# B&R Automation Studio project Embraco_LinkaNaOdlievanieRotorov_DokoncovaciaStanica_Rev2
Automation Studio 4.10.3.60 SP; technology packages: Acp10Arnc0 5.15.1, mapp 5.15.0

## Configuration Config1

CPU X20cPS9400, AutomationRuntime B4.91, Build 6.3.0, Safety 1.10, Vc V4.72.6

### Task classes (Cpu.sw)
```
Cyclic#1 (cycle 3000 us, tolerance 0 us):
  RychleDeje <- Program.RychleDeje.prg
  VstupnyMan <- Program.VstupnyManipulator.prg
Cyclic#2 (cycle 10000 us, tolerance 10000 us):
  RiadenieSe <- RiadenieServ.RiadenieServ.prg
  Serva_Prir <- RiadenieServ.Serva_PriradenieVstupov.prg
  StanicaVa1 <- Program.StanicaVonkajsiehoValcovania.prg
  StanicaStr <- Program.StanicaStrihania.prg
  StanicaVal <- Program.StanicaVnutornehoValcovania.prg
  StanicaMer <- Program.StanicaMerania.prg
  RiadenieMe <- RiadenieMenicov.RiadenieMenicov.prg
  Blikanie10 <- Blikace.Blikanie10ms.prg
Cyclic#3:
  Blikanie1 <- Blikace.Blikanie50ms.prg
  OtocnyStol <- Program.OtocnyStol.prg
Cyclic#4 (cycle 200000 us, tolerance 200000 us):
  Blikanie20 <- Blikace.Blikanie200ms.prg
  ZdvihRotor <- Program.ZdvihRotora.prg
Cyclic#5 (cycle 500000 us, tolerance 500000 us):
  Blikanie50 <- Blikace.Blikanie500ms.prg
Cyclic#6 (cycle 1000000 us, tolerance 1000000 us):
  Blikanie1s <- Blikace.Blikanie1s.prg
Cyclic#7 (cycle 5000000 us, tolerance 5000000 us):
  Blikanie5s <- Blikace.Blikanie5s.prg
Cyclic#8 (cycle 100000 us, tolerance 100000 us):
  VystupnyOd <- Program.VystupnyOdsuvac.prg
  StanicaRaz <- Program.StanicaRazenia.prg
  VystupnyMa <- Program.VystupnyManipulator.prg
  Oddelovac <- Program.Oddelovac.prg
  Main <- Program.Main.prg
  Komunikaci <- Komunikacia.KOM_HlavnaLinka.prg
  Poruchy_Si <- Program.Poruchy_Signalizacie.prg
DataObjects: Acp10sys, assl1
NcDataObjects: acp10etxen <- RiadenieServ.acp10etxen.dob, gAxis01a <- RiadenieServ.VstupnyManipulator.gAxis01a.dob, gAxis01i <- RiadenieServ.VstupnyManipulator.gAxis01i.dob, gAxis02a <- RiadenieServ.VystupnyManipulator.gAxis02a.dob, gAxis02i <- RiadenieServ.VystupnyManipulator.gAxis02i.dob, gAxis03a <- RiadenieServ.ZdvihValcovacky.gAxis03a.dob, gAxis03i <- RiadenieServ.ZdvihValcovacky.gAxis03i.dob, gAxis04a <- RiadenieServ.ZdvihRotora.gAxis04a.dob, gAxis04i <- RiadenieServ.ZdvihRotora.gAxis04i.dob
VcDataObjects: Visu <- Vizualizacia.Visu.dob
Binaries: udbdef, TCData, arsvcreg, vccbtn, arialbd, vcmgr, vcgclass, vcfile, vccnum, vctcal, vcdsloc, vcbclass, vcfntttf, vccalarm, arial, vcpdi815, vccshape, vcalarm, vcptelo, Visu01, vccdt, vcpdsw, vcpdihd, vcpk, vccbmp, vccstr, vcpfppc7, vcrt, vcshared, Visu02, vcctext, vcclbox, vccbar, vcpdi855, vcdsint, vccovl, vccline, Visu03, iomap, asfw, Role, ashwac, sysconf, Config_1, ashwd, Config, User, arconfig, acp10cfg, Acp10map, vcchspot
Libraries: Acp10par, NcGlobal, Acp10man, AsSafety, FileIO, DataObj, AsXml, standard, runtime, astime, AsEPL, AsIOAcc, Acp10_MC, brsystem, sys_lib, IecCheck, SC, AsBrStr, MpRecipe, MpBase, AxisLib, asieccon, powerlnk, vcresman
```

### Hardware
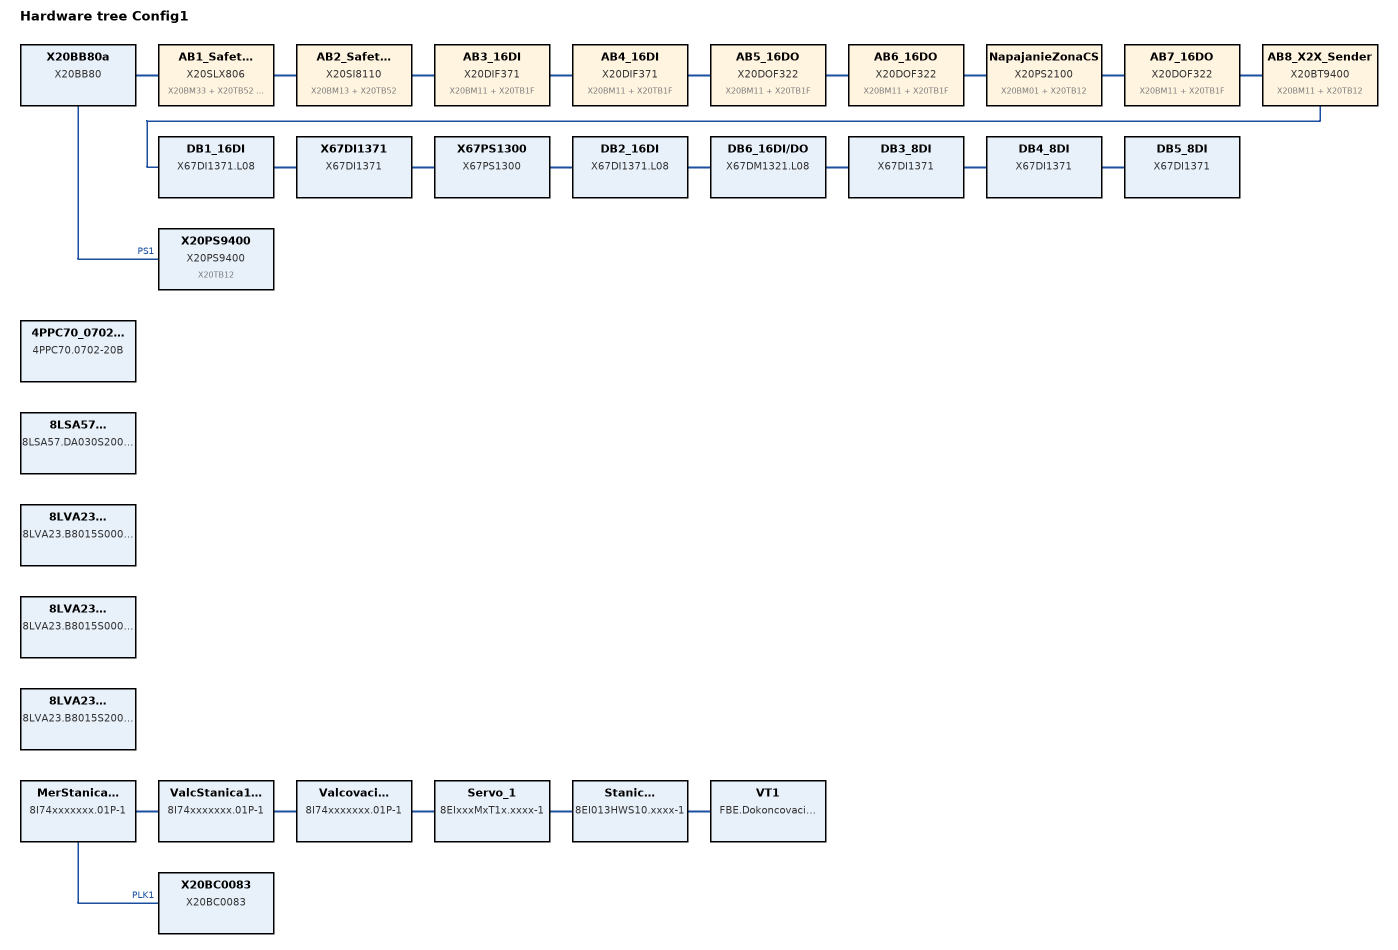
```
4PPC70_0702_20B : 4PPC70.0702-20B v1.5.4.0
  Connector IF1:
    DNAConfiguration = manual
    CycleTime = 1000
    EplNatSubnet = 192.168.100.0
  Connector IF2:
    ActivateDevice = 1
    Mode = Manual
    InternetAddress = 192.168.0.3
    SubnetMask = 255.255.255.0
    ActivateModbus = 1
    NumSlaves = -1
    NumAllBlocks = -1
    MemSizeIn = -1
    MemSizeOut = -1
    ModbusSlaveGrey = 1
    ModbusSlaveConfig_1
    InputRegisterChannelGroup1_1
    InputRegisterChannelID1_1 = OUT_1
    InputRegisterChannelType1_1 = UINT
    InputRegisterChannelGroup2_1
    InputRegisterChannelID2_1 = OUT_2
    InputRegisterChannelAddress2_1 = 8193
    InputRegisterChannelType2_1 = UINT
    InputRegisterChannelGroup3_1
    InputRegisterChannelID3_1 = OUT_3
    InputRegisterChannelAddress3_1 = 8194
    InputRegisterChannelType3_1 = UINT
    InputRegisterChannelGroup4_1
    InputRegisterChannelID4_1 = OUT_4
    InputRegisterChannelAddress4_1 = 8195
    InputRegisterChannelType4_1 = UINT
    InputRegisterChannelGroup5_1
    InputRegisterChannelID5_1 = OUT_5
    InputRegisterChannelAddress5_1 = 8196
    InputRegisterChannelType5_1 = UINT
    HoldingRegisterChannelGroup1_1
    HoldingRegisterChannelID1_1 = IN_1
    HoldingRegisterChannelType1_1 = UINT
    HoldingRegisterChannelGroup2_1
    HoldingRegisterChannelID2_1 = IN_2
    HoldingRegisterChannelAddress2_1 = 24577
    HoldingRegisterChannelType2_1 = UINT
    HoldingRegisterChannelGroup3_1
    HoldingRegisterChannelID3_1 = IN_3
    HoldingRegisterChannelAddress3_1 = 24578
    HoldingRegisterChannelType3_1 = UINT
    HoldingRegisterChannelGroup4_1
    HoldingRegisterChannelID4_1 = IN_4
    HoldingRegisterChannelAddress4_1 = 24579
    HoldingRegisterChannelType4_1 = UINT
    HoldingRegisterChannelGroup5_1
    HoldingRegisterChannelID5_1 = IN_5
    HoldingRegisterChannelAddress5_1 = 24580
    HoldingRegisterChannelType5_1 = UINT
    ModbusMaster = 0
  Connector IF5:
    CycleTime = 1000
  ConfigurationID = Embraco_LinkaNaOdlievanieRotorov_DokoncovaciaStanica_Config1
  UserPartitionSize = 0
  PermanentPvSize = 2000
  RemanentGlobalPvSize = 2000
  DisableProfiling = 1
  TimerDeviceType = EPLX2X
  TimerDevice = 4PPC70_0702_20B.IF1
  TaskClassIdleTime = 2000
  Cyclic1Duration = 3000
  Cyclic1Tolerance = 0
  Cyclic2Duration = 10000
  Cyclic2Tolerance = 10000
  Cyclic4Duration = 200000
  Cyclic4Tolerance = 200000
  Cyclic5Duration = 500000
  Cyclic5Tolerance = 500000
  Cyclic6Duration = 1000000
  Cyclic6Tolerance = 1000000
  Cyclic7Duration = 5000000
  Cyclic7Tolerance = 5000000
  Cyclic8Duration = 100000
  Cyclic8Tolerance = 100000
  FileDevice1
  FileDeviceName1 = HDD
  FileDevicePath1 = C:\
  TimeZone = 145
  FtpUser1
  FtpUsername1 = admin
  FtpUserPassword1 = kfejnbuok6+6ErbPl2VMIFPsI8vTqz8wcboRfqSMuVU=
  FtpUserSalt1 = 0YUTbZnu
  FTPAccessRight1 = 0
  FTPMSPartition1 = SYSTEM
  VcObjectName = Visu
  KeyMappingFile = VC\4PPC70_0702_20B.dis
8LSA57.DA030S200-3 : 8LSA57.DA030S200-3 v1.0.5.34  [EC -> StanicaValcovania2.EC1; MT -> StanicaValcovania2.MT1]
8LVA23.B8015S000-0 : 8LVA23.B8015S000-0 v1.0.1.30  [EC -> Servo_1.EC1; MT -> Servo_1.MT1]
8LVA23.B8015S000-0a : 8LVA23.B8015S000-0 v1.0.1.30  [EC -> Servo_1.EC2; MT -> Servo_1.MT2]
8LVA23.B8015S200-0 : 8LVA23.B8015S200-0 v2.2.0.3  [EC -> Servo_1.EC3; MT -> Servo_1.MT3]
AB1_SafetyMaster : X20SLX806 v1.10.12.1  [SS1 -> X20TB52.SS; SS2 -> X20TB52a.SS; SL -> X20BM33.SL1]
  Supervision = off
  SafeProject = SafeLOGIC-1
  SafeDesigner = 4.3.4.4
  DigitalOutput01 = viaSafeLOGIC
  DigitalOutput02 = viaSafeLOGIC
  DigitalOutput03 = viaSafeLOGIC
  DigitalOutput04 = viaSafeLOGIC
  DigitalOutput05 = viaSafeLOGIC
  DigitalOutput06 = viaSafeLOGIC
  UnsafeOutputBOOLs = 16
  UnsafeInputBOOLs = 16
AB2_SafetyInputs : X20SI8110 v1.10.12.0  [SS1 -> X20TB52b.SS; SL -> X20BM13.SL1]
  Supervision = off
AB3_16DI : X20DIF371 v1.2.0.0  [SS1 -> X20TB1F.SS; SL -> X20BM11.SL1]
  Supervision = off
AB4_16DI : X20DIF371 v1.2.0.0  [SS1 -> X20TB1F1.SS; SL -> X20BM11a.SL1]
  Supervision = off
AB5_16DO : X20DOF322 v1.5.0.0  [SS1 -> X20TB1F2.SS; SL -> X20BM11b.SL1]
  Supervision = off
AB6_16DO : X20DOF322 v1.5.0.0  [SS1 -> X20TB1F4.SS; SL -> X20BM11e.SL1]
  Supervision = off
AB7_16DO : X20DOF322 v1.5.0.0  [SS1 -> X20TB1F3.SS; SL -> X20BM11c.SL1]
  Supervision = off
AB8_X2X_Sender : X20BT9400 v1.3.0.0  [SS1 -> X20TB12b.SS; SL -> X20BM11d.SL1]
  Supervision = off
  PowerInfo = on
DB1_16DI : X67DI1371.L08 v1.1.0.0  [X2X1 -> AB8_X2X_Sender.X2X1 [Cable Type=X2XCable, Length=10, Version=1.0.0.3]]
  Supervision = off
DB2_16DI : X67DI1371.L08 v1.1.0.0  [X2X1 -> X67PS1300.X2X2 [Cable Type=X2XCable, Length=10, Version=1.0.0.3]]
  Supervision = off
DB3_8DI : X67DI1371 v1.1.0.0  [X2X1 -> DB6_16DI/DO.X2X2 [Cable Type=X2XCable, Length=10, Version=1.0.0.3]]
  Supervision = off
DB4_8DI : X67DI1371 v1.1.0.0  [X2X1 -> DB3_8DI.X2X2 [Cable Type=X2XCable, Length=10, Version=1.0.0.3]]
  Supervision = off
DB5_8DI : X67DI1371 v1.1.0.0  [X2X1 -> DB4_8DI.X2X2 [Cable Type=X2XCable, Length=10, Version=1.0.0.3]]
  Supervision = off
DB6_16DI/DO : X67DM1321.L08 v1.3.0.0  [X2X1 -> DB2_16DI.X2X2 [Cable Type=X2XCable, Length=10, Version=1.0.0.3]]
  Supervision = off
  Direction14 = output
  Direction15 = output
  Direction16 = output
MerStanica_OtacanieRotora : 8I74xxxxxxx.01P-1 v1.6.2.0  [PLK1 -> X20BC0083.PLK1 [Cable Type=PowerlinkCable, Length=10, Version=1.0.0.3]; PLK2 -> ValcStanica1_OtacanieRotora.PLK1 [Cable Type=PowerlinkCable, Length=10, Version=1.0.0.3]]
  FunctionModel = Standard
  Supervision = off
  LFRD_LFR_Filter = LFR_RFR
  ACC = 10
  DEC = 10
  CTT = 0
  NPR = 25
  COS = 77
  UNS = 230
  NCR = 13
  NSP = 1380
  PTCL = 1
NapajanieZonaCS : X20PS2100 v1.4.0.0  [SS1 -> X20TB12a.SS; SL -> X20BM01.SL1]
  Supervision = off
  PowerInfo = on
Servo_1 : 8EIxxxMxT1x.xxxx-1 v2.3.1.1  [PLK1 -> ValcovaciaStanica2_OtacanieNastroja.PLK2 (NodeNumber=4) [Cable Type=PowerlinkCable, Length=10, Version=1.0.0.3]; PLK2 -> StanicaValcovania2.PLK1 (NodeNumber=4) [Cable Type=PowerlinkCable, Length=10, Version=1.0.0.3]; EC1 -> 8LVA23.B8015S000-0.EC; EC2 -> 8LVA23.B8015S000-0a.EC; EC3 -> 8LVA23.B8015S200-0.EC; MT2 -> 8LVA23.B8015S000-0a.MT; MT3 -> 8LVA23.B8015S200-0.MT]
  BothEndSwitchesAreNormallyOpen_r1 = on
  QuickStopIsNormallyOpen_r1 = on
  BothEndSwitchesAreNormallyOpen_r2 = on
  QuickStopIsNormallyOpen_r2 = on
  BothEndSwitchesAreNormallyOpen_r3 = on
  QuickStopIsNormallyOpen_r3 = on
  Ax1Interface = Ax1EnDat
  Ax2Interface = Ax2EnDat
  Ax3Interface = Ax3EnDat
StanicaValcovania2 : 8EI013HWS10.xxxx-1 v2.3.1.1  [PLK1 -> Servo_1.PLK2 (NodeNumber=7) [Cable Type=PowerlinkCable, Length=10, Version=1.0.0.3]; PLK2 -> VT1.PLK1 (NodeNumber=7) [Cable Type=PowerlinkCable, Length=10, Version=1.0.0.3]; EC1 -> 8LSA57.DA030S200-3.EC]
  MotionTP = Acp10Arnc0
  BothEndSwitchesAreNormallyOpen_r1 = on
  QuickStopIsNormallyOpen_r1 = on
  Ax1Interface = Ax1EnDat
VT1 : FBE.DokoncovaciaStanica_VT1 v11.13.09 (OrderNumber=VT1)  [PLK1 -> StanicaValcovania2.PLK2 (NodeNumber=5) [Cable Type=PowerlinkCable, Length=10, Version=1.0.0.3]]
  Supervision = off
  p2000s01_direction = wo
  p2000s02_direction = wo
  p2000s03_direction = wo
  p2000s04_direction = wo
ValcStanica1_OtacanieRotora : 8I74xxxxxxx.01P-1 v1.6.2.0  [PLK1 -> MerStanica_OtacanieRotora.PLK2 [Cable Type=PowerlinkCable, Length=10, Version=1.0.0.3]; PLK2 -> ValcovaciaStanica2_OtacanieNastroja.PLK1 [Cable Type=PowerlinkCable, Length=10, Version=1.0.0.3]]
  FunctionModel = Standard
  Supervision = off
  LFRD_LFR_Filter = LFR_RFR
  ACC = 10
  DEC = 10
  CTT = 0
  NPR = 150
  COS = 79
  UNS = 230
  NCR = 56
  NSP = 1415
  PTCL = 1
ValcovaciaStanica2_OtacanieNastroja : 8I74xxxxxxx.01P-1 v1.6.2.0  [PLK1 -> ValcStanica1_OtacanieRotora.PLK2 (NodeNumber=6) [Cable Type=PowerlinkCable, Length=10, Version=1.0.0.3]; PLK2 -> Servo_1.PLK1 (NodeNumber=6) [Cable Type=PowerlinkCable, Length=10, Version=1.0.0.3]]
  FunctionModel = Standard
  Supervision = off
  LFRD_LFR_Filter = LFR_RFR
  ACC = 40
  DEC = 40
  CTT = 0
  NPR = 110
  COS = 84
  UNS = 400
  NCR = 25
  NSP = 2825
  BLC = 2
  PTCL = 1
X20BB80a : X20BB80 v1.1.0.0
X20BC0083 : X20BC0083 v2.14.0.0  [PLK1 -> MerStanica_OtacanieRotora.PLK1 [Cable Type=PowerlinkCable, Length=10, Version=1.0.0.3]; PLK2 -> 4PPC70_0702_20B.IF1 [Cable Type=PowerlinkCable, Length=10, Version=1.0.0.3]; SL -> X20BB80a.SL1]
  Supervision = off
X20BM01 : X20BM01 v2.2.0.0  [X2X1 -> X20BM11e.X2X2]
X20BM11 : X20BM11 v1.1.0.0  [X2X1 -> X20BM13.X2X2]
X20BM11a : X20BM11 v1.1.0.0  [X2X1 -> X20BM11.X2X2]
X20BM11b : X20BM11 v1.1.0.0  [X2X1 -> X20BM11a.X2X2]
X20BM11c : X20BM11 v1.1.0.0  [X2X1 -> X20BM01.X2X2]
X20BM11d : X20BM11 v1.1.0.0  [X2X1 -> X20BM11c.X2X2]
X20BM11e : X20BM11 v1.1.0.0  [X2X1 -> X20BM11b.X2X2]
X20BM13 : X20BM13 v1.1.0.0  [X2X1 -> X20BM33.X2X2]
X20BM33 : X20BM33 v1.1.0.0  [X2X1 -> X20BB80a.IF1]
X20PS9400 : X20PS9400 v1.7.0.0  [SS1 -> X20TB12c.SS; PS -> X20BB80a.PS1]
  Supervision = off
  PowerInfo = on
X20TB12a : X20TB12 v1.0.0.0
X20TB12b : X20TB12 v1.0.0.0
X20TB12c : X20TB12 v1.0.0.0
X20TB1F : X20TB1F v1.0.0.0
X20TB1F1 : X20TB1F v1.0.0.0
X20TB1F2 : X20TB1F v1.0.0.0
X20TB1F3 : X20TB1F v1.0.0.0
X20TB1F4 : X20TB1F v1.0.0.0
X20TB52 : X20TB52 v1.0.0.2
X20TB52a : X20TB52 v1.0.0.2
X20TB52b : X20TB52 v1.0.0.2
X67DI1371 : X67DI1371 v1.1.0.0  [X2X1 -> DB1_16DI.X2X2 [Cable Type=X2XCable, Length=10, Version=1.0.0.3]]
  Supervision = off
X67PS1300 : X67PS1300 v1.0.0.0  [X2X1 -> X67DI1371.X2X2 [Cable Type=X2XCable, Length=10, Version=1.0.0.3]]
```

### Cpu.per - 4PPC70_0702_20B/Cpu.per
```iecst
VAR_CONFIG
	Valcovanie_RychlostJog_MM_s AT %MD0; (* *)
	VstupManipul_RychlostJog_MM_s AT %MD4; (* *)
	VystupManipul_RychlostJog_MM_s AT %MD8; (* *)
	Stol_Pozicia_1 AT %MB12; (*Pozicia stola pod meranim  0 - neznamy kus, 1 - kus OK, 2 - kus NG *)
	Stol_Pozicia_2 AT %MB13; (*Pozícia medzi meranim a výstupným manipulátorom    0 - neznamy kus, 1 - kus OK, 2 - kus NG *)
	Stol_Pozicia_3 AT %MB14; (*Pozícia pod výstupným manipulátorom     0 - neznamy kus, 1 - kus OK, 2 - kus NG *)
	TP_Meranie_CasMerania AT %MD16; (*v s*)
	TP_Meranie_RychlostOtacania AT %MW20; (*v Hz*)
	TP_Razenie_CasRazenia AT %MD24; (*v s*)
	TP_Valcovanie_PoziciaVnorenia AT %MD28; (*v mm*)
	TP_Valcovanie_RychlostOtacania AT %MW32; (*v Hz*)
	TP_Valcovanie_RychlostZdvihu AT %MD36; (*v mm/s*)
	TP_VstupManip_PoziciaOdoberania AT %MD40; (*v mm*)
	TP_VstupManip_PoziciaUkladania AT %MD44; (*v mm*)
	TP_VstupManip_RychlostPojazdu AT %MD48; (*v mm/s*)
	TP_VystupManip_PoziciaOdoberania AT %MD52; (*v mm*)
	TP_VystupManip_PoziciaUklad_NG AT %MD56; (*v mm*)
	TP_VystupManip_PoziciaUklad_OK AT %MD60; (*v mm*)
	TP_VystupManip_RychlostPojazdu AT %MD64; (*v mm/s*)
	TP_Valcovanie_CasStrekuOleja AT %MD68; (*v s*)
	TP_Valcovanie_PocetCyklPredStrek AT %MW72; (* *)
	VstupManipulator_Drzi_NG_Kus AT %MX74; (* *)
	TP_CasValcovania_s AT %MD76; (*v sek*)
	Valcovanie2_CasValcovania_s AT %MD80; (* *)
	Valcovanie2_FM_DobehRampa_s AT %MD84; (* *)
	Valcovanie2_FM_RozbehRampa_s AT %MD88; (* *)
	Valcovanie2_FM_RychlostOtac_Hz AT %MD92; (* *)
	Valcovanie2_ServoJoggRychl_MM_s AT %MD96; (* *)
	Valcovanie2_ServoPracRychl1_MM_s AT %MD100; (* *)
	Valcovanie2_ServoPracRychl2_MM_s AT %MD104; (* *)
	Valcovanie2_CasStrekuOleja_s AT %MD108; (* *)
	Valcovanie2_MomentPritlaku_Nm AT %MD112; (* *)
	Valcovanie2_PocetCyklStrekuOleja AT %MB116; (* *)
	Valcovanie2_ZadanaPozMM AT %MD120; (* *)
	Valcovanie2_ZadanaPozSTART_MM AT %MD124; (*Čakacia pozícia pod stolom*)
END_VAR
```

### IoMap.iom - 4PPC70_0702_20B/IoMap.iom
```iecst
VAR_CONFIG
	Cyclic#1.siCS_KanalA AT %IX."AB1_SafetyMaster".SafeDigitalInput01;
	Cyclic#1.siCS_KanalB AT %IX."AB1_SafetyMaster".SafeDigitalInput02;
	Cyclic#1.siServisneDvere1_KanalA AT %IX."AB1_SafetyMaster".SafeDigitalInput03;
	Cyclic#1.siServisneDvere1_KanalB AT %IX."AB1_SafetyMaster".SafeDigitalInput04;
	Cyclic#1.siServisneDvere2_KanalA AT %IX."AB1_SafetyMaster".SafeDigitalInput05;
	Cyclic#1.siServisneDvere2_KanalB AT %IX."AB1_SafetyMaster".SafeDigitalInput06;
	Cyclic#1.siServisneDvere3_KanalA AT %IX."AB1_SafetyMaster".SafeDigitalInput07;
	Cyclic#1.siServisneDvere3_KanalB AT %IX."AB1_SafetyMaster".SafeDigitalInput08;
	Cyclic#1.siServisneDvere4_KanalA AT %IX."AB2_SafetyInputs".SafeDigitalInput01;
	Cyclic#1.siServisneDvere4_KanalB AT %IX."AB2_SafetyInputs".SafeDigitalInput02;
	Cyclic#1.siServisneDvere5_KanalA AT %IX."AB2_SafetyInputs".SafeDigitalInput03;
	Cyclic#1.siServisneDvere5_KanalB AT %IX."AB2_SafetyInputs".SafeDigitalInput04;
	Cyclic#1.soMotory AT %IX."AB1_SafetyMaster".PhysicalStateChannel01;
	Cyclic#1.soVystupy AT %IX."AB1_SafetyMaster".PhysicalStateChannel02;
	Cyclic#1.soKomunikacia_StavCS AT %IX."AB1_SafetyMaster".PhysicalStateChannel03;
	Cyclic#1.Reset_CS AT %QX."AB1_SafetyMaster".BOOL101;
	Cyclic#1.Reset_Oplotenia AT %QX."AB1_SafetyMaster".BOOL102;
	Cyclic#1.Stav_BZ5_Zamknuty AT %IX."AB1_SafetyMaster".BOOL007;
	Cyclic#1.Stav_BZ4_Zamknuty AT %IX."AB1_SafetyMaster".BOOL006;
	Cyclic#1.Stav_BZ3_Zamknuty AT %IX."AB1_SafetyMaster".BOOL005;
	Cyclic#1.Stav_BZ2_Zamknuty AT %IX."AB1_SafetyMaster".BOOL004;
	Cyclic#1.Stav_BZ1_Zamknuty AT %IX."AB1_SafetyMaster".BOOL003;
	Cyclic#1.Stav_CS_Odblokovane AT %IX."AB1_SafetyMaster".BOOL002;
	Cyclic#1.SafetyPLC_Nabehlo AT %IX."AB1_SafetyMaster".BOOL001;
	Cyclic#1.diStav_PrivodVzduchuKanalA AT %QX."AB1_SafetyMaster".BOOL103;
	Cyclic#1.diStav_PrivodVzduchuKanalB AT %QX."AB1_SafetyMaster".BOOL104;
	Cyclic#1.diStavReleKA100_KA101 AT %QX."AB1_SafetyMaster".BOOL105;
	Cyclic#1.diStavReleKA102_KA103 AT %QX."AB1_SafetyMaster".BOOL106;
	Cyclic#1.diStavReleKA104_KA105 AT %QX."AB1_SafetyMaster".BOOL107;
	Cyclic#1.BezpOkruhOplotenia_Aktivovany AT %IX."AB1_SafetyMaster".BOOL010;
	Cyclic#1.BezpOkruhCS_Aktivovany AT %IX."AB1_SafetyMaster".BOOL009;
	Cyclic#1.Stav_BZ6_Zamknuty AT %IX."AB1_SafetyMaster".BOOL008;
	Cyclic#1.siServisneDvere6_KanalA AT %IX."AB2_SafetyInputs".SafeDigitalInput05;
	Cyclic#1.siServisneDvere6_KanalB AT %IX."AB2_SafetyInputs".SafeDigitalInput06;
	Cyclic#1.diMeranie_PoruchaOtacRotora AT %IX."AB3_16DI".DigitalInput01;
	Cyclic#1.diValcovanie_PoruchaOtacRotora AT %IX."AB3_16DI".DigitalInput02;
	Cyclic#1.diStol_PoruchaOtacStola AT %IX."AB3_16DI".DigitalInput03;
	Cyclic#1.diStol_TeplotaMotoraOK AT %IX."AB3_16DI".DigitalInput04;
	Cyclic#1.diPoruchaNapajaniaSERVO1 AT %IX."AB3_16DI".DigitalInput05;
	Cyclic#1.diHydraulika_PoruchaCerpadla AT %IX."AB3_16DI".DigitalInput06;
	Cyclic#1.diBZ1_DvereZavrete AT %IX."AB3_16DI".DigitalInput09;
	Cyclic#1.diBZ2_DvereZavrete AT %IX."AB3_16DI".DigitalInput10;
	Cyclic#1.diBZ3_DvereZavrete AT %IX."AB3_16DI".DigitalInput11;
	Cyclic#1.diBZ4_DvereZavrete AT %IX."AB3_16DI".DigitalInput12;
	Cyclic#1.diBZ5_DvereZavrete AT %IX."AB3_16DI".DigitalInput13;
	Cyclic#1.diStavReleKA100_KA101 AT %IX."AB3_16DI".DigitalInput14;
	Cyclic#1.diStavReleKA102_KA103 AT %IX."AB3_16DI".DigitalInput15;
	Cyclic#1.diStavReleKA104_KA105 AT %IX."AB3_16DI".DigitalInput16;
	Cyclic#1.diStav_PrivodVzduchuKanalA AT %IX."AB4_16DI".DigitalInput01;
	Cyclic#1.diStav_PrivodVzduchuKanalB AT %IX."AB4_16DI".DigitalInput02;
	Cyclic#1.diBZ6_DvereZavrete AT %IX."AB4_16DI".DigitalInput03;
	Cyclic#1.doHydraulika_ChodCerpadla AT %QX."AB5_16DO".DigitalOutput01;
	Cyclic#1.doBZ1_ZamkniZamok AT %QX."AB5_16DO".DigitalOutput02;
	Cyclic#1.doBZ2_ZamkniZamok AT %QX."AB5_16DO".DigitalOutput03;
	Cyclic#1.doBZ3_ZamkniZamok AT %QX."AB5_16DO".DigitalOutput04;
	Cyclic#1.doBZ4_ZamkniZamok AT %QX."AB5_16DO".DigitalOutput05;
	Cyclic#1.doBZ5_ZamkniZamok AT %QX."AB5_16DO".DigitalOutput06;
	Cyclic#1.doValcovanie_DavkaOleja AT %QX."AB5_16DO".DigitalOutput07;
	Cyclic#1.doKontrolkaPORUCHA AT %QX."AB5_16DO".DigitalOutput08;
	Cyclic#1.doMajak_CerveneSvetlo AT %QX."AB5_16DO".DigitalOutput09;
	Cyclic#1.doMajak_ZlteSvetlo AT %QX."AB5_16DO".DigitalOutput10;
	Cyclic#1.doMajak_ZeleneSvetlo AT %QX."AB5_16DO".DigitalOutput11;
	Cyclic#1.doMajak_Hukacka AT %QX."AB5_16DO".DigitalOutput12;
	Cyclic#1.doStol_ResetPoruchy AT %QX."AB5_16DO".DigitalOutput13;
	Cyclic#1.doBZ6_ZamkniZamok AT %QX."AB5_16DO".DigitalOutput14;
	Cyclic#1.doRazenie_ZdvihRotora AT %QX."AB7_16DO".DigitalOutput01;
	Cyclic#1.doRazenie_ZostupRotora AT %QX."AB7_16DO".DigitalOutput02;
	Cyclic#1.Vyrazanie.OUT.VyrazanieVysunut AT %QX."AB7_16DO".DigitalOutput03;
	Cyclic#1.Vyrazanie.OUT.VyrazanieZasunut AT %QX."AB7_16DO".DigitalOutput04;
	Cyclic#1.doStol_OtacajVPRED AT %QX."AB7_16DO".DigitalOutput05;
	Cyclic#1.doStol_OtacajVZAD AT %QX."AB7_16DO".DigitalOutput06;
	Cyclic#1.doStol_ODBRZDENIE AT %QX."AB7_16DO".DigitalOutput07;
	Cyclic#1.diStol_SnimacPolohyStola AT %IX."DB1_16DI".DigitalInput01;
	Cyclic#1.Vyrazanie.IN.KusPritomny AT %IX."DB1_16DI".DigitalInput02;
	Cyclic#1.Vyrazanie.IN.VyrazanieJeDole AT %IX."DB1_16DI".DigitalInput03;
	Cyclic#1.Vyrazanie.IN.VyrazanieJeHore AT %IX."DB1_16DI".DigitalInput04;
	Cyclic#1.Vyrazanie.IN.CentrovanieZatvorene AT %IX."DB1_16DI".DigitalInput05;
	Cyclic#1.Vyrazanie.IN.CentrovanieOtvorene AT %IX."DB1_16DI".DigitalInput06;
	Cyclic#1.Vyrazanie.IN.UchytenieKolikaDrzimkus AT %IX."DB1_16DI".DigitalInput07;
	Cyclic#1.Vyrazanie.IN.UchytenieNaliatkuDrzimkus AT %IX."DB1_16DI".DigitalInput08;
	Cyclic#1.Vyrazanie.IN.OdhadzovanieJeVzadu AT %IX."DB1_16DI".DigitalInput09;
	Cyclic#1.Vyrazanie.IN.OdhadzovanieJeVpredu AT %IX."DB1_16DI".DigitalInput10;
	Cyclic#1.diRazenie_ZdvihSpodnaPoloha AT %IX."DB1_16DI".DigitalInput11;
	Cyclic#1.diValcovanie_PritomnostRotora AT %IX."DB2_16DI".DigitalInput03;
	Cyclic#1.diValcovanie_GriperOtvoreny AT %IX."DB2_16DI".DigitalInput04;
	Cyclic#1.diValcovanie_GriperZatvoreny AT %IX."DB2_16DI".DigitalInput05;
	Cyclic#1.diValcovanie_HladinaOlejaOK AT %IX."DB2_16DI".DigitalInput06;
	Cyclic#1.diMeranie_ZdvihSpodnaPoloha AT %IX."DB2_16DI".DigitalInput09;
	Cyclic#1.diMeranie_ZdvihHornaPoloha AT %IX."DB2_16DI".DigitalInput10;
	Cyclic#1.diMeranie_PritomnostRotora AT %IX."DB2_16DI".DigitalInput11;
	Cyclic#1.diStol_PritomnostRotoraVstup AT %IX."DB2_16DI".DigitalInput15;
	Cyclic#1.diStol_PritomnostRotoraVystup AT %IX."DB2_16DI".DigitalInput16;
	Cyclic#1.diVstupManipul_ZasunutyHore AT %IX."DB3_8DI".DigitalInput01;
	Cyclic#1.diVstupManipul_VysunutyDole AT %IX."DB3_8DI".DigitalInput02;
	Cyclic#1.diVstupManipul_PrednyLimitSnimac AT %IX."DB3_8DI".DigitalInput03 INVERSE;
	Cyclic#1.diVstupManipul_ZadnyLimitSnimac AT %IX."DB3_8DI".DigitalInput04 INVERSE;
	Cyclic#1.diVystupManipul_ZasunutyHore AT %IX."DB4_8DI".DigitalInput01;
	Cyclic#1.diVystupManipul_PrednyLimSnimac AT %IX."DB4_8DI".DigitalInput03 INVERSE;
	Cyclic#1.diVystupManipul_ZadnyLimSnimac AT %IX."DB4_8DI".DigitalInput04 INVERSE;
	Cyclic#1.doOddelovac_PrepniPozNavazania AT %QX."VT1".Valve_1_C14;
	Cyclic#1.doOddelovac_PrepniPozVyvazania AT %QX."VT1".Valve_1_C12;
	Cyclic#1.doVystupManipul_GriperZATVOR AT %QX."VT1".Valve_5_C14;
	Cyclic#1.doVystupManipul_GriperOTVOR AT %QX."VT1".Valve_5_C12;
	Cyclic#1.doVystDopr_OdsuvacVYSUN AT %QX."VT1".Valve_6_C14;
	Cyclic#1.doVystDopr_OdsuvacZASUN AT %QX."VT1".Valve_6_C12;
	Cyclic#1.Vyrazanie.OUT.OdhadzovanieVysunut AT %QX."VT1".Valve_9_C14;
	Cyclic#1.Vyrazanie.OUT.OdhadzovanieZasunut AT %QX."VT1".Valve_9_C12;
	Cyclic#1.::FM_Menic[1].IO.ModuleOk AT %IX."MerStanica_OtacanieRotora".ModuleOk;
	Cyclic#1.::FM_Menic[1].IO.ReadyToSwitchOn AT %IX."MerStanica_OtacanieRotora".ETAD_Input_Bool_00;
	Cyclic#1.::FM_Menic[1].IO.SwitchedOn AT %IX."MerStanica_OtacanieRotora".ETAD_Input_Bool_01;
	Cyclic#1.::FM_Menic[1].IO.Running AT %IX."MerStanica_OtacanieRotora".ETAD_Input_Bool_02;
	Cyclic#1.::FM_Menic[1].IO.Fault AT %IX."MerStanica_OtacanieRotora".ETAD_Input_Bool_03;
	Cyclic#1.::FM_Menic[1].IO.VoltageEnabled AT %IX."MerStanica_OtacanieRotora".ETAD_Input_Bool_04;
	Cyclic#1.::FM_Menic[1].IO.SwitchOnDisabled AT %IX."MerStanica_OtacanieRotora".ETAD_Input_Bool_06;
	Cyclic#1.::FM_Menic[1].IO.StavRiadeniaMenica AT %IX."MerStanica_OtacanieRotora".ETAD_Input_Bool_09;
	Cyclic#1.::FM_Menic[1].IO.PoziciaDosiahnuta AT %IX."MerStanica_OtacanieRotora".ETAD_Input_Bool_10;
	Cyclic#1.::FM_Menic[1].IO.SmerOtacania AT %IX."MerStanica_OtacanieRotora".ETAD_Input_Bool_15;
	Cyclic#1.::FM_Menic[1].IO.ErrorNumber AT %IW."MerStanica_OtacanieRotora".LFT_Input;
	Cyclic#1.::FM_Menic[1].IO.SwitchOn AT %QX."MerStanica_OtacanieRotora".CMDD_Output_Bool_00;
	Cyclic#1.::FM_Menic[1].IO.DisableVoltage AT %QX."MerStanica_OtacanieRotora".CMDD_Output_Bool_01;
	Cyclic#1.::FM_Menic[1].IO.QuickStop AT %QX."MerStanica_OtacanieRotora".CMDD_Output_Bool_02;
	Cyclic#1.::FM_Menic[1].IO.Run AT %QX."MerStanica_OtacanieRotora".CMDD_Output_Bool_03;
	Cyclic#1.::FM_Menic[1].IO.FaultReset AT %QX."MerStanica_OtacanieRotora".CMDD_Output_Bool_07;
	Cyclic#1.::FM_Menic[1].IO.Direction AT %QX."MerStanica_OtacanieRotora".CMDD_Output_Bool_11;
	Cyclic#1.::FM_Menic[1].IO.SpeedSetpoint AT %QW."MerStanica_OtacanieRotora".LFR_Output;
	Cyclic#1.::FM_Menic[1].IO.OutputFrequency AT %IW."MerStanica_OtacanieRotora".RFR_Input;
	Cyclic#1.::FM_Menic[1].IO.MotorTorque AT %IW."MerStanica_OtacanieRotora".OTR_Input;
	Cyclic#1.::FM_Menic[1].IO.MotorCurrent AT %IW."MerStanica_OtacanieRotora".LCR_Input;
	Cyclic#1.::FM_Menic[2].IO.ModuleOk AT %IX."ValcStanica1_OtacanieRotora".ModuleOk;
	Cyclic#1.::FM_Menic[2].IO.ReadyToSwitchOn AT %IX."ValcStanica1_OtacanieRotora".ETAD_Input_Bool_00;
	Cyclic#1.::FM_Menic[2].IO.SwitchedOn AT %IX."ValcStanica1_OtacanieRotora".ETAD_Input_Bool_01;
	Cyclic#1.::FM_Menic[2].IO.Running AT %IX."ValcStanica1_OtacanieRotora".ETAD_Input_Bool_02;
	Cyclic#1.::FM_Menic[2].IO.Fault AT %IX."ValcStanica1_OtacanieRotora".ETAD_Input_Bool_03;
	Cyclic#1.::FM_Menic[2].IO.VoltageEnabled AT %IX."ValcStanica1_OtacanieRotora".ETAD_Input_Bool_04;
	Cyclic#1.::FM_Menic[2].IO.SwitchOnDisabled AT %IX."ValcStanica1_OtacanieRotora".ETAD_Input_Bool_06;
	Cyclic#1.::FM_Menic[2].IO.StavRiadeniaMenica AT %IX."ValcStanica1_OtacanieRotora".ETAD_Input_Bool_09;
	Cyclic#1.::FM_Menic[2].IO.PoziciaDosiahnuta AT %IX."ValcStanica1_OtacanieRotora".ETAD_Input_Bool_10;
	Cyclic#1.::FM_Menic[2].IO.SmerOtacania AT %IX."ValcStanica1_OtacanieRotora".ETAD_Input_Bool_15;
	Cyclic#1.::FM_Menic[2].IO.ErrorNumber AT %IW."ValcStanica1_OtacanieRotora".LFT_Input;
	Cyclic#1.::FM_Menic[2].IO.SwitchOn AT %QX."ValcStanica1_OtacanieRotora".CMDD_Output_Bool_00;
	Cyclic#1.::FM_Menic[2].IO.DisableVoltage AT %QX."ValcStanica1_OtacanieRotora".CMDD_Output_Bool_01;
	Cyclic#1.::FM_Menic[2].IO.QuickStop AT %QX."ValcStanica1_OtacanieRotora".CMDD_Output_Bool_02;
	Cyclic#1.::FM_Menic[2].IO.Run AT %QX."ValcStanica1_OtacanieRotora".CMDD_Output_Bool_03;
	Cyclic#1.::FM_Menic[2].IO.FaultReset AT %QX."ValcStanica1_OtacanieRotora".CMDD_Output_Bool_07;
	Cyclic#1.::FM_Menic[2].IO.Direction AT %QX."ValcStanica1_OtacanieRotora".CMDD_Output_Bool_11;
	Cyclic#1.::FM_Menic[2].IO.SpeedSetpoint AT %QW."ValcStanica1_OtacanieRotora".LFR_Output;
	Cyclic#1.::FM_Menic[2].IO.OutputFrequency AT %IW."ValcStanica1_OtacanieRotora".RFR_Input;
	Cyclic#1.::FM_Menic[2].IO.MotorTorque AT %IW."ValcStanica1_OtacanieRotora".OTR_Input;
	Cyclic#1.::FM_Menic[2].IO.MotorCurrent AT %IW."ValcStanica1_OtacanieRotora".LCR_Input;
	Cyclic#1.doValcovanie_ZDVIH_Rotora AT %QX."VT1".Valve_10_C14;
	Cyclic#1.doValcovanie_ZOSTUP_Rotora AT %QX."VT1".Valve_10_C12;
	Cyclic#1.doMeranie_ZDVIH AT %QX."VT1".Valve_12_C14;
	Cyclic#1.doMeranie_ZOSTUP AT %QX."VT1".Valve_12_C12;
	Cyclic#1.diVstupManipul_ZdvihStredPoloha AT %IX."DB3_8DI".DigitalInput07;
	Cyclic#1.diRazenie_PritomnostRotora AT %IX."DB1_16DI".DigitalInput12;
	Cyclic#1.diRazenie_ZdvihHornaPoloha AT %IX."DB1_16DI".DigitalInput13;
	Cyclic#1.diValcovanie_ZdvihHornaPoloha AT %IX."DB2_16DI".DigitalInput07;
	Cyclic#1.diValcovanie_ZdvihSpodnaPoloha AT %IX."DB2_16DI".DigitalInput08;
	Cyclic#1.diVystupManipul_ZdvihStredPoloha AT %IX."DB4_8DI".DigitalInput02;
	Cyclic#1.diVystupManipul_VysunutyDole AT %IX."DB4_8DI".DigitalInput07;
	Cyclic#1.::diVystDopr_OdsuvacZasunuty AT %IX."DB5_8DI".DigitalInput03;
	Cyclic#1.::diVystDopr_OdsuvacVysunuty AT %IX."DB5_8DI".DigitalInput04;
	Cyclic#1.::diOddelovac_PritomnostRotora AT %IX."DB5_8DI".DigitalInput06;
	Cyclic#1.::diOddelovac_PoziciaNavazanie AT %IX."DB5_8DI".DigitalInput07;
	Cyclic#1.::diOddelovac_PoziciaVyvazanie AT %IX."DB5_8DI".DigitalInput08;
	Cyclic#1.diVstupDopr_PritomnostRotora AT %IX."DB5_8DI".DigitalInput05;
	Cyclic#1.diHydraulika_Stav_FilterZaneseny AT %IX."AB4_16DI".DigitalInput04;
	Cyclic#1.doLEDosvetlenie_ZeleneSvetlo AT %QX."AB6_16DO".DigitalOutput01;
	Cyclic#1.doLEDosvetlenie_CerveneSvetlo AT %QX."AB6_16DO".DigitalOutput02;
	Cyclic#1.doLEDosvetlenie_ModreSvetlo AT %QX."AB6_16DO".DigitalOutput03;
	Cyclic#1.doLEDosvetlenie_BieleSvetlo AT %QX."AB6_16DO".DigitalOutput04;
	Cyclic#1.doValcovanie_GriperZATVOR AT %QX."VT1".Valve_11_C14;
	Cyclic#1.doValcovanie_GriperOTVOR AT %QX."VT1".Valve_11_C12;
	Cyclic#1.doVstupManipul_ZOSTUP AT %QX."VT1".Valve_2_C14;
	Cyclic#1.doVstupManipul_ZDVIH AT %QX."VT1".Valve_2_C12;
	Cyclic#1.doVstupManipul_GriperZATVOR AT %QX."VT1".Valve_3_C12;
	Cyclic#1.doVstupManipul_GriperOTVOR AT %QX."VT1".Valve_3_C14;
	Cyclic#1.doVystupManipul_ZDVIH AT %QX."VT1".Valve_4_C12;
	Cyclic#1.doVystupManipul_ZOSTUP AT %QX."VT1".Valve_4_C14;
	Cyclic#1.Vyrazanie.OUT.UchytenieNaliatkuOtvorit AT %QX."VT1".Valve_7_C14;
	Cyclic#1.Vyrazanie.OUT.UchytenieNaliatkuZatvorit AT %QX."VT1".Valve_7_C12;
	Cyclic#1.Vyrazanie.OUT.UchytenieKolikaOtvorit AT %QX."VT1".Valve_8_C14;
	Cyclic#1.Vyrazanie.OUT.UchytenieKolikaZatvorit AT %QX."VT1".Valve_8_C12;
	Cyclic#1.diValcovanie_HornyLimitSnimac AT %IX."DB2_16DI".DigitalInput02 INVERSE;
	Cyclic#1.diValcovanie_SpodnyLimitSnimac AT %IX."DB2_16DI".DigitalInput01 INVERSE;
	Cyclic#1.diTlacitko_RotorOK AT %IX."AB4_16DI".DigitalInput05;
	Cyclic#1.diTlacitko_RotorNG AT %IX."AB4_16DI".DigitalInput06;
	Cyclic#1.doCervenaLED_Tlacitko_rotor_NG AT %QX."AB5_16DO".DigitalOutput16;
	Cyclic#1.doZelenaLED_Tlacitko_rotor_OK AT %QX."AB5_16DO".DigitalOutput15;
	Cyclic#1.diVstupManipul_GriperOtvoreny AT %IX."DB3_8DI".DigitalInput06;
	Cyclic#1.diVstupManipul_GriperZatvoreny AT %IX."DB3_8DI".DigitalInput05;
	Cyclic#1.diValcovanie_PritomnostNastroja AT %IX."DB2_16DI".DigitalInput14;
	Cyclic#1.diVystupManipul_GriperZatvoreny AT %IX."DB4_8DI".DigitalInput05;
	Cyclic#1.diVystupManipul_GriperOtvoreny AT %IX."DB4_8DI".DigitalInput06;
	Cyclic#1.::diHlavnyPrivodVzduchu_TlakOK AT %IX."AB4_16DI".DigitalInput16;
	Cyclic#1.::RezimServis AT %QX."AB1_SafetyMaster".BOOL108;
	Cyclic#1.ModBus_Output1 AT %QW."4PPC70_0702_20B".IF2.OUT_1;
	Cyclic#1.ModBus_Output2 AT %QW."4PPC70_0702_20B".IF2.OUT_2;
	Cyclic#1.ModBus_Output3 AT %QW."4PPC70_0702_20B".IF2.OUT_3;
	Cyclic#1.ModBus_Output4 AT %QW."4PPC70_0702_20B".IF2.OUT_4;
	Cyclic#1.ModBus_Output5 AT %QW."4PPC70_0702_20B".IF2.OUT_5;
	Cyclic#1.ModBus_Input1 AT %IW."4PPC70_0702_20B".IF2.IN_1;
	Cyclic#1.ModBus_Input2 AT %IW."4PPC70_0702_20B".IF2.IN_2;
	Cyclic#1.ModBus_Input3 AT %IW."4PPC70_0702_20B".IF2.IN_3;
	Cyclic#1.ModBus_Input4 AT %IW."4PPC70_0702_20B".IF2.IN_4;
	Cyclic#1.ModBus_Input5 AT %IW."4PPC70_0702_20B".IF2.IN_5;
	Cyclic#1.doZatvorenieOdvzdHydrauliky AT %QX."AB6_16DO".DigitalOutput05;
	Cyclic#1.doVstupDopr_VysunZdvihRotora AT %QX."VT1".Valve_13_C14;
	Cyclic#1.diVstupDopr_ZdvihRotora_HORE AT %IX."DB1_16DI".DigitalInput15;
	Cyclic#1.diVstupDopr_ZdvihRotora_DOLE AT %IX."DB1_16DI".DigitalInput14;
	Cyclic#1.diHydraulika_TeplotaOlejaOK AT %IX."AB3_16DI".DigitalInput07;
	Cyclic#1.diHydraulika_HladinaOlejaOK AT %IX."AB3_16DI".DigitalInput08;
	Cyclic#1.diVstupManipul_HornSnimacNG_Kusu AT %IX."DB3_8DI".DigitalInput08;
	Cyclic#1.diVstupManipul_SpodSnimacNG_Kusu AT %IX."DB4_8DI".DigitalInput08;
	Cyclic#1.::FM_Menic[3].IO.ModuleOk AT %IX."ValcovaciaStanica2_OtacanieNastroja".ModuleOk;
	Cyclic#1.::FM_Menic[3].IO.ReadyToSwitchOn AT %IX."ValcovaciaStanica2_OtacanieNastroja".ETAD_Input_Bool_00;
	Cyclic#1.::FM_Menic[3].IO.SwitchedOn AT %IX."ValcovaciaStanica2_OtacanieNastroja".ETAD_Input_Bool_01;
	Cyclic#1.::FM_Menic[3].IO.Running AT %IX."ValcovaciaStanica2_OtacanieNastroja".ETAD_Input_Bool_02;
	Cyclic#1.::FM_Menic[3].IO.Fault AT %IX."ValcovaciaStanica2_OtacanieNastroja".ETAD_Input_Bool_03;
	Cyclic#1.::FM_Menic[3].IO.VoltageEnabled AT %IX."ValcovaciaStanica2_OtacanieNastroja".ETAD_Input_Bool_04;
	Cyclic#1.::FM_Menic[3].IO.SwitchOnDisabled AT %IX."ValcovaciaStanica2_OtacanieNastroja".ETAD_Input_Bool_06;
	Cyclic#1.::FM_Menic[3].IO.StavRiadeniaMenica AT %IX."ValcovaciaStanica2_OtacanieNastroja".ETAD_Input_Bool_09;
	Cyclic#1.::FM_Menic[3].IO.PoziciaDosiahnuta AT %IX."ValcovaciaStanica2_OtacanieNastroja".ETAD_Input_Bool_10;
	Cyclic#1.::FM_Menic[3].IO.SmerOtacania AT %IX."ValcovaciaStanica2_OtacanieNastroja".ETAD_Input_Bool_15;
	Cyclic#1.::FM_Menic[3].IO.ErrorNumber AT %IW."ValcovaciaStanica2_OtacanieNastroja".LFT_Input;
	Cyclic#1.::FM_Menic[3].IO.SwitchOn AT %QX."ValcovaciaStanica2_OtacanieNastroja".CMDD_Output_Bool_00;
	Cyclic#1.::FM_Menic[3].IO.DisableVoltage AT %QX."ValcovaciaStanica2_OtacanieNastroja".CMDD_Output_Bool_01;
	Cyclic#1.::FM_Menic[3].IO.QuickStop AT %QX."ValcovaciaStanica2_OtacanieNastroja".CMDD_Output_Bool_02;
	Cyclic#1.::FM_Menic[3].IO.Run AT %QX."ValcovaciaStanica2_OtacanieNastroja".CMDD_Output_Bool_03;
	Cyclic#1.::FM_Menic[3].IO.FaultReset AT %QX."ValcovaciaStanica2_OtacanieNastroja".CMDD_Output_Bool_07;
	Cyclic#1.::FM_Menic[3].IO.Direction AT %QX."ValcovaciaStanica2_OtacanieNastroja".CMDD_Output_Bool_11;
	Cyclic#1.::FM_Menic[3].IO.SpeedSetpoint AT %QW."ValcovaciaStanica2_OtacanieNastroja".LFR_Output;
	Cyclic#1.::FM_Menic[3].IO.OutputFrequency AT %IW."ValcovaciaStanica2_OtacanieNastroja".RFR_Input;
	Cyclic#1.::FM_Menic[3].IO.MotorTorque AT %IW."ValcovaciaStanica2_OtacanieNastroja".OTR_Input;
	Cyclic#1.::FM_Menic[3].IO.MotorCurrent AT %IW."ValcovaciaStanica2_OtacanieNastroja".LCR_Input;
	Cyclic#1.::Modul_DB1_OK AT %IX."DB1_16DI".ModuleOk;
	Cyclic#1.::Modul_DB2_OK AT %IX."DB2_16DI".ModuleOk;
	Cyclic#1.::Modul_DB3_OK AT %IX."DB3_8DI".ModuleOk;
	Cyclic#1.::Modul_DB4_OK AT %IX."DB4_8DI".ModuleOk;
	Cyclic#1.::Modul_DB5_OK AT %IX."DB5_8DI".ModuleOk;
	Cyclic#1.::Modul_DB6_OK AT %IX."DB6_16DI/DO".ModuleOk;
	Cyclic#1.diValc2_TlakPritlaku_OK AT %IX."DB6_16DI/DO".DigitalInput01;
	Cyclic#1.diValc2_PritomnostRotora AT %IX."DB6_16DI/DO".DigitalInput02;
	Cyclic#1.diValc2_SpomalenieZdvihu AT %IX."DB6_16DI/DO".DigitalInput03;
	Cyclic#1.diValc2_PritlakZasunuty AT %IX."DB6_16DI/DO".DigitalInput04;
	Cyclic#1.diValc2_PritlakVysunuty AT %IX."DB6_16DI/DO".DigitalInput05;
	Cyclic#1.diValc2_ZdvihSpodnyLimit AT %IX."DB6_16DI/DO".DigitalInput06;
	Cyclic#1.diValc2_ZdvihHornyLimit AT %IX."DB6_16DI/DO".DigitalInput07;
	Cyclic#1.doValc2_DavkaOleja AT %QX."DB6_16DI/DO".DigitalOutput14;
	Cyclic#1.diValc2_PorMotoraOtacania AT %IX."AB4_16DI".DigitalInput07;
	Cyclic#1.diValc2_PorNapajaniaServa AT %IX."AB4_16DI".DigitalInput08;
	Cyclic#1.diValc2_OdbrzdOtacNastrojaMenic AT %IX."AB4_16DI".DigitalInput09;
	Cyclic#1.doValc2_BrzdaOtacNastroja AT %QX."AB6_16DO".DigitalOutput06;
	Cyclic#1.diValc2_ZdvihRotoraZasunuty AT %IX."DB6_16DI/DO".DigitalInput08;
	Cyclic#1.diValc2_OdbrzdOtacNastrojaRuka AT %IX."DB6_16DI/DO".DigitalInput09;
	Cyclic#1.diValc2_SnimacOtacaniaNastroja AT %IX."DB6_16DI/DO".DigitalInput10;
	Cyclic#1.doValc2_ZdvihPritlakuHORE AT %QX."AB6_16DO".DigitalOutput08;
	Cyclic#1.doValc2_ZostupPritlakuDOLE AT %QX."AB6_16DO".DigitalOutput07;
	Cyclic#1.diMeranie_Osciloskop_Stav_OK AT %IX."AB4_16DI".DigitalInput10;
	Cyclic#1.diMeranie_Osciloskop_Stav_NG AT %IX."AB4_16DI".DigitalInput11;
	Cyclic#1.doMeranie_Osciloskop_START AT %QX."AB6_16DO".DigitalOutput09;
	Cyclic#1.doMeranie_Osciloskop_STOP AT %QX."AB6_16DO".DigitalOutput10;
	Cyclic#1.doMeranie_Osciloskop_Frekvencia AT %QX."AB6_16DO".DigitalOutput16;
	Cyclic#1.diVystDoprOK_SnimacZaplnTrate AT %IX."DB5_8DI".DigitalInput02;
	Cyclic#1.diVystDoprNG_SnimacZaplnTrate AT %IX."DB5_8DI".DigitalInput01;
	Cyclic#1.Vyrazanie.IN.KusOstalPrilepeny AT %IX."X67DI1371".DigitalInput01;
	Cyclic#1.Vyrazanie.IN.UchytenieNaliatkuZatvorene AT %IX."X67DI1371".DigitalInput02;
	Cyclic#1.Vyrazanie.IN.UchytenieNaliatkuOtvorene AT %IX."X67DI1371".DigitalInput03;
	Cyclic#1.Stol.IN.CentrovanieVysunute AT %IX."X67DI1371".DigitalInput05;
	Cyclic#1.Stol.IN.CentrovanieZasunute AT %IX."X67DI1371".DigitalInput06;
	Cyclic#1.Vyrazanie.IN.UchytenieKolikaZatvorene AT %IX."X67DI1371".DigitalInput07;
	Cyclic#1.Vyrazanie.IN.UchytenieKolikaOtvorene AT %IX."X67DI1371".DigitalInput08;
	Cyclic#1.Vyrazanie.IN.OdhadzovanieJeVpredu2 AT %IX."X67DI1371".DigitalInput04;
	Cyclic#1.Vyrazanie.OUT.CentrovanieZatvorit AT %QX."VT1".Valve_15_C12;
	Cyclic#1.Vyrazanie.OUT.CentrovanieOtvorit AT %QX."VT1".Valve_15_C14;
	Cyclic#1.Stol.OUT.CentrovanieZasunut AT %QX."VT1".Valve_14_C14;
	Cyclic#1.Stol.OUT.CentrovanieVysunut AT %QX."VT1".Valve_14_C12;
	Cyclic#1.diStol_NaliatokOdstrihnuty  AT %IX."DB1_16DI".DigitalInput16 INVERSE;
END_VAR
```

### Acp10cfg.ncc - 4PPC70_0702_20B/Motion/Acp10cfg.ncc
```
NcConfiguration (Version=5.00.2, NcSwId=Acp10)
  ACP10CF1_typ:
    cnt_nettrc_rec_drive = 150
    bufsize_trace_upload = 1200
    tc_nc_man_task = Cyclic #1
    glob_pv_as_ncobject = Yes
    ncsys_dl_broadcast = Yes
    ncsys_dl_acp_reset = Yes
    safemc_log_err_to_ax = Yes
    network_init:
      ncsw_init_execute = Yes
      automatic_execute = No
      node_nr_warning = Yes
      net_err_before_ncact = Yes
    nettrc:
      enter_parsecrec = Yes
      enter_ncaction = Yes
      save_ring_startidx = No
    cam_prof_download:
      cam_dat_dl_parallel = No
      tc_cam_dl_parallel = Task class for NC Manager task
    plk_if[0]:
      if_name = IF1
      tc_CycDat_PLCopen = Task class for NC Manager task
      mc_broadcast_extdat = No
```

### Acp10map.ncm - 4PPC70_0702_20B/Motion/Acp10map.ncm
```
NcMapping (NcSwId=Acp10)
  NcObject gAxis01 (ModuleId=Servo_1, Type=ncAXIS, Channel=1, AcoposSimulation=Off, InitParameter=gAxis01i, AcoposParameter=gAxis01a, Disabled=FALSE, ModuleDisabled=FALSE)
  NcObject gAxis02 (ModuleId=Servo_1, Type=ncAXIS, Channel=2, AcoposSimulation=Off, InitParameter=gAxis02i, AcoposParameter=gAxis02a, Disabled=FALSE, ModuleDisabled=FALSE)
  NcObject gAxis03 (ModuleId=Servo_1, Type=ncAXIS, Channel=3, AcoposSimulation=Off, InitParameter=gAxis03i, AcoposParameter=gAxis03a, Disabled=FALSE, ModuleDisabled=FALSE)
  NcObject 8EIxxxMxT1x.xxxx-1_ncV_AXIS1 (ModuleId=Servo_1, Type=ncV_AXIS, Channel=1, Disabled=TRUE, ModuleDisabled=FALSE)
  NcObject 8EIxxxMxT1x.xxxx-1_ncV_AXIS2 (ModuleId=Servo_1, Type=ncV_AXIS, Channel=2, Disabled=TRUE, ModuleDisabled=FALSE)
  NcObject 8EIxxxMxT1x.xxxx-1_ncV_AXIS3 (ModuleId=Servo_1, Type=ncV_AXIS, Channel=3, Disabled=TRUE, ModuleDisabled=FALSE)
  NcObject gAxis04 (ModuleId=StanicaValcovania2, Type=ncAXIS, Channel=1, AcoposSimulation=Off, InitParameter=gAxis04i, AcoposParameter=gAxis04a, Disabled=FALSE, ModuleDisabled=FALSE)
  NcObject 8EI013HWS10.xxxx-1_ncV_AXIS1 (ModuleId=StanicaValcovania2, Type=ncV_AXIS, Channel=1, Disabled=TRUE, ModuleDisabled=FALSE)
```

- Safety project (password-protected, skipped)

### Config.mprecipexml - 4PPC70_0702_20B/mappServices/Config.mprecipexml
```
Element gRecipeXmlLink (Type=mprecipexml)
```

### Config_1.mprecipexml - 4PPC70_0702_20B/mappServices/Config_1.mprecipexml
```
Element gRecipeUzivatelXmlLink (Type=mprecipexml)
```

## Logical view

Binary libraries used (declarations not repeated): operator, runtime, astime, AsIecCon, AsSafety, FileIO, DataObj, AsXml, standard, AsEPL, AsIOAcc, brsystem, sys_lib, AsBrStr, Acp10man 5.15.1, Acp10par 5.15.1, NcGlobal 5.15.1, Acp10_MC 5.15.1, MpRecipe 5.15.0, MpBase 5.15.0

### Global.typ - Global data types
```iecst
TYPE
	InverterTypes :
		( (*Possible inverter types*)
		X64 := 1,
		P74 := 2,
		P84 := 3
		);
	INVERTER_STATES :
		(
		INVERTER_WAIT, (*Wait for command*)
		INVERTER_RUN, (*State where the inverter is running with set speed*)
		INVERTER_POWER_ON, (*Power on the inverter*)
		INVERTER_POWER_OFF, (*Power off the inverter*)
		INVERTER_TUNE_X64, (*Autotune the inverter.*)
		INVERTER_TUNE_P74, (*Autotune the inverter.*)
		INVERTER_TUNE_P84, (*Autotune the inverter.*)
		INVERTER_STOP, (*Stop the movement*)
		INVERTER_ERROR (*Error state*)
		);
	InverterInputCommand_typ : 	STRUCT
		AutoTune : BOOL; (*Command to autotune the inverter, It will be turned on for 2sec during this operation*)
		RunForward : BOOL; (*Run with positive direction. *)
		Acknowledge : BOOL;
		RunBackward : BOOL; (*Run with negative direction. *)
		RunLowSpeed : BOOL; (*Run with lowspeed. If lowspeed is false, highspeed will be used.*)
	END_STRUCT;
	InverterInput_typ : 	STRUCT
		Command : InverterInputCommand_typ; (*Command structure*)
		LowSpeed : INT; (*Set lowspeed*)
		HighSpeed : INT; (*Set highspeed*)
		AccTime : UINT; (*Acceleration time to nominal frequency in 0.1s*)
		DecTime : UINT; (*Deceleration time from nominal frequency 0.1s*)
		DeviceString : STRING[80]; (*The device adress used. Eg *IF6.ST2*. Is needed to write parameters.*)
		InverterType : InverterTypes; (*Type of B&R inverter. X64, P74 or P84.*)
		Node : USINT; (*Powerlink node number of the inverter. Only required when inverter type is P74 or P84.*)
		StopType : USINT; (*0 = Stop by stop command bit. 1 = stop by setting the spedsetpoint to 0. *)
		InverterName : STRING[80]; (*Name of the inverter, not required.*)
	END_STRUCT;
	InverterOutputStatus_typ : 	STRUCT
		Error : BOOL; (*An error occured, see ErrorNumber*)
		ErrorText : STRING[80]; (*Inverter error text*)
		ErrorNumber : UINT; (*Error number for additional information*)
		Tuned : BOOL;
		Running : BOOL;
	END_STRUCT;
	InverterOutput_typ : 	STRUCT
		Status : InverterOutputStatus_typ; (*Status information*)
	END_STRUCT;
	Inverter_typ : 	STRUCT
		Input : InverterInput_typ; (*Input structure*)
		Output : InverterOutput_typ; (*Output structure*)
		State : INVERTER_STATES; (*States of the state machine*)
		SubState : UINT; (*Substates*)
		IO : Inverter_IO_typ; (*IO structure to be mapped to the inverter IO mapping*)
	END_STRUCT;
END_TYPE

(*The IO structure is only used for the inverter IO mapping*)

TYPE
	Error_Info_typ : 	STRUCT
		ErrorText : ARRAY[0..110]OF STRING[100]; (*Text info about possible faults*)
	END_STRUCT;
	Inverter_IO_typ : 	STRUCT
		ModuleOk : BOOL; (*Module okay status*)
		SwitchOn : BOOL; (*Swith on the inverter command*)
		Run : BOOL; (*Command RUN*)
		SpeedSetpoint : INT; (*Speed setpoint to the inverter*)
		ReadyToSwitchOn : BOOL; (*Status that the inverter is ready to switch on*)
		SwitchedOn : BOOL; (*Status that the inverter is switched on*)
		Running : BOOL; (*Status that the inverter is running*)
		Fault : BOOL; (*Status that a fault have accoured*)
		ErrorNumber : INT; (*The error number in case of an inverter error*)
		FaultReset : BOOL; (*Fault reset command*)
		Stop : BOOL; (*Stop command. Not currently used in this task. The speed setpoint is set to 0 instead.*)
		Direction : BOOL; (*Direction of rotation*)
		Decelerating : BOOL; (*Status when the inverter is decelerating*)
		Brake : BOOL; (*Mapped to R2 if a brake funktion is needed*)
		TargetReached : BOOL; (*Status when the speed setpoint is reached*)
		SpeedMode : BOOL; (*Status when the inverter is running*)
		OutputFrequency : INT; (*Output frequency of the inverter*)
		MotorCurrent : UINT; (*Output current of the inverter*)
		MotorTorque : INT; (*Output torque of the inverter*)
		SwitchOnDisabled : BOOL; (*Status*)
		VoltageEnabled : BOOL; (*Status*)
		DisableVoltage : BOOL; (*Command Disable Voltage*)
		QuickStop : BOOL; (*Command Quick Stop*)
		StavRiadeniaMenica : BOOL; (*Status  0 - riadený z panela, 1- riadený cez komunikáciu*)
		PoziciaDosiahnuta : BOOL; (*Status*)
		SmerOtacania : BOOL; (*Status 0 - smer dopredu, 1 - smer dozadu*)
	END_STRUCT;
END_TYPE

(***************Uzivatelia****************************)

TYPE
	ParametreUzivatelovTyp : 	STRUCT
		Meno : STRING[50];
		Heslo : STRING[50];
		UrovenUzivatela : UINT;
	END_STRUCT;
END_TYPE

(************Receptury*************************)

TYPE
	ParametreRecepturTyp : 	STRUCT
		Nazov : STRING[30];
		Premenna_1 : REAL;
		Premenna_2 : REAL;
		Premenna_3 : USINT;
		Premenna_4 : USINT;
		Premenna_5 : USINT;
		Premenna_6 : USINT;
	END_STRUCT;
END_TYPE

(************Dorobok cani*************************)

TYPE
	StolStruc : 	STRUCT
		OUT : StolOUT;
		IN : StolIN;
	END_STRUCT;
	VyrazanieStruc : 	STRUCT
		OUT : VyrazanieOUT;
		IN : VyrazanieIN;
	END_STRUCT;
	StolOUT : 	STRUCT
		CentrovanieZasunut : BOOL;
		CentrovanieVysunut : BOOL;
	END_STRUCT;
	VyrazanieOUT : 	STRUCT
		VyrazanieZasunut : BOOL;
		VyrazanieVysunut : BOOL;
		OdhadzovanieZasunut : BOOL;
		OdhadzovanieVysunut : BOOL;
		CentrovanieZatvorit : BOOL;
		CentrovanieOtvorit : BOOL;
		UchytenieNaliatkuOtvorit : BOOL;
		UchytenieNaliatkuZatvorit : BOOL;
		UchytenieKolikaOtvorit : BOOL;
		UchytenieKolikaZatvorit : BOOL;
	END_STRUCT;
	StolIN : 	STRUCT
		CentrovanieZasunute : BOOL;
		CentrovanieVysunute : BOOL;
	END_STRUCT;
	VyrazanieIN : 	STRUCT
		KusPritomny : BOOL;
		KusOstalPrilepeny : BOOL;
		CentrovanieOtvorene : BOOL;
		UchytenieKolikaZatvorene : BOOL;
		UchytenieNaliatkuDrzimkus : BOOL;
		VyrazanieJeHore : BOOL;
		CentrovanieZatvorene : BOOL;
		OdhadzovanieJeVpredu2 : BOOL;
		OdhadzovanieJeVpredu : BOOL;
		UchytenieKolikaOtvorene : BOOL;
		UchytenieNaliatkuZatvorene : BOOL;
		UchytenieNaliatkuOtvorene : BOOL;
		OdhadzovanieJeVzadu : BOOL;
		UchytenieKolikaDrzimkus : BOOL;
		VyrazanieJeDole : BOOL;
	END_STRUCT;
END_TYPE
```

### Global.var - Global variables
```iecst
(*************Premenne receptur**************)
VAR
	SC_Uzivatelia : SequenceControlTyp;
	MpRecipeRegPar_0 : MpRecipeRegPar := (0);
	MpRecipeXml_0 : MpRecipeXml := (0);
	Receptura : ARRAY[0..20] OF ParametreRecepturTyp := [21((0))];
	UlozRecepturu : BOOL := FALSE;
	NacitajRecepturu : BOOL;
	Nazov : STRING[30] := '';
	Premenna_1 : REAL;
	Premenna_2 : REAL;
	Premenna_3 : USINT;
	Premenna_4 : USINT;
	Premenna_5 : USINT;
	Premenna_6 : USINT;
	ZvolenyNazovProduktu : STRING[30];
	ZvolenaPremenna_1 : REAL;
	ZvolenaPremenna_2 : REAL;
	ZvolenaPremenna_3 : USINT;
	ZvolenaPremenna_4 : USINT;
	ZvolenaPremenna_5 : USINT;
	ZvolenaPremenna_6 : USINT;
END_VAR
(**********Premenne uzivatelov********************************)
VAR
	MpRecipeXml_1 : MpRecipeXml := (0);
	MpRecipeRegPar_1 : MpRecipeRegPar := (0);
	Uzivatel : ARRAY[0..20] OF ParametreUzivatelovTyp;
	ZoznamUzivatelov : ARRAY[0..20] OF STRING[50] := [21('')];
	MenoUzivatela : STRING[50];
	HesloUzivatela : STRING[50];
	UrovenUzivatela : UINT;
	ZadaneMenoUzivatela : STRING[50];
	ZadaneHesloUzivatela : STRING[50];
	ZvolenyUzivatel : STRING[50];
	ZvolenaUroven : UINT;
	TP_ZobrazPopUpPrihlasenie : USINT;
	UlozUzivatelov : BOOL;
	PrihlasUzivatela : BOOL;
	VymazUzivatela : BOOL;
	OdhlasUzivatela : BOOL;
END_VAR
(**********Blikače*******************************)
VAR
	Blikac200ms : BOOL;
	Blikac500ms : BOOL;
	Blikac1s : BOOL;
	Blikac5s : BOOL;
	Blikac50ms : BOOL;
	Blikac10ms : BOOL;
END_VAR
(*********RiadenieServ*************************)
VAR
	gAxis01 : ACP10AXIS_typ;
	gAxis02 : ACP10AXIS_typ;
	gAxis03 : ACP10AXIS_typ;
	gAxis04 : ACP10AXIS_typ;
	Motion : ARRAY[1..4] OF Axis;
	idx : USINT := 0;
END_VAR
VAR CONSTANT
	MAX_MOTION : USINT := 4;
END_VAR
VAR
	Servo1_PriradenieSnimacov : MC_BR_SetHardwareInputs;
	Servo2_PriradenieSnimacov : MC_BR_SetHardwareInputs;
	Servo3_PriradenieSnimacov : MC_BR_SetHardwareInputs;
	Servo4_PriradenieSnimacov : MC_BR_SetHardwareInputs;
END_VAR
(************Riadenie FM meničov*********************)
VAR
	ErrorInfo : ARRAY[1..2] OF Error_Info_typ;
END_VAR
VAR CONSTANT
	NR_OF_INVERTERS : USINT := 3;
END_VAR
VAR
	FM_Menic : ARRAY[1..NR_OF_INVERTERS] OF Inverter_typ;
END_VAR
(*************Safety premenné*****************************)
VAR
	RezimServis : BOOL;
	SafetyPLC_Nabehlo : BOOL;
	BezpOkruhCS_Aktivovany : BOOL;
	BezpOkruhOplotenia_Aktivovany : BOOL;
	Reset_CS : BOOL;
	Reset_Oplotenia : BOOL;
	Stav_CS_Odblokovane : BOOL;
	Stav_BZ1_Zamknuty : BOOL;
	Stav_BZ2_Zamknuty : BOOL;
	Stav_BZ3_Zamknuty : BOOL;
	Stav_BZ4_Zamknuty : BOOL;
	Stav_BZ5_Zamknuty : BOOL;
	Stav_BZ6_Zamknuty : BOOL;
	Zamkni_BZ1 : BOOL;
	Zamkni_BZ2 : BOOL;
	Zamkni_BZ3 : BOOL;
	Zamkni_BZ4 : BOOL;
	Zamkni_BZ5 : BOOL;
	Zamkni_BZ6 : BOOL;
	StavZamkuBZ1 : USINT;
	StavZamkuBZ2 : USINT;
	StavZamkuBZ3 : USINT;
	StavZamkuBZ4 : USINT;
	StavZamkuBZ5 : USINT;
	StavZamkuBZ6 : USINT;
END_VAR
(*********Meranie prestojov********************)
VAR
	StratovyCas_START : BOOL;
	StratovyCas_Milisekundy : UINT;
	StratovyCas_Sekundy : UINT;
	StratovyCas_Minuty : UINT;
	StratovyCas_Hodiny : UINT;
	StratovyCas_RESET : BOOL;
END_VAR
(*****************Alarmy*************************)
VAR
	Alarmy : ARRAY[0..100] OF BOOL;
	NastalaPorucha : BOOL;
	ZobrazSymbolAlarmu : BOOL;
	PotvrdenieAlarmov : BOOL;
	PoruchaOddelovaca : BOOL;
	PoruchaZdvihuRotora : BOOL;
	PoruchaVstupManipulator : BOOL;
	PoruchaOtocnyStol : BOOL;
	PoruchaStanicaStrihania : BOOL;
	PoruchaStanicaRazenia : BOOL;
	PoruchaStanicaValcovania : BOOL;
	PoruchaStanicaValcovania2 : BOOL;
	PoruchaStanicaMerania : BOOL;
	PoruchaVystupManipulator : BOOL;
	PoruchaVystupOdsuvac : BOOL;
	VypnutieHukacky : BOOL;
END_VAR
(************Všeobecné premenné************)
VAR
	Modul_DB1_OK : BOOL;
	Modul_DB2_OK : BOOL;
	Modul_DB3_OK : BOOL;
	Modul_DB4_OK : BOOL;
	Modul_DB5_OK : BOOL;
	Modul_DB6_OK : BOOL;
	Zariadenie_Moduly_OK : BOOL;
	Zariadenie_TaktTime : REAL;
	Zariadenie_Automat : BOOL;
	Zariadenie_Manual : BOOL;
	Zariadenie_Reset : BOOL;
	Zariadenie_PoINIT : BOOL;
	Zariadenie_HOME : BOOL;
	Zariadenie_KoniecVyroby : BOOL;
	Zariadenie_KoniecCyklu : BOOL;
	Zariadenie_RevorkRezim : BOOL;
	Zariadenie_StavAutomat : BOOL;
	Zariadenie_StavManual : BOOL;
	Zariadenie_StavPoINIT : BOOL;
	Zariadenie_HomingOK : BOOL;
	Zariadenie_PrebiehaHoming : BOOL;
	Zariadenie_PrebiehaUkoncenie : BOOL;
	Zariadenie_PrebiehaKoniecCyklu : BOOL;
	Zariadenie_PrebiehaRevorkRezim : BOOL;
	Zariadenie_PAUZA : BOOL;
	VnutorneValcovanie_AKTIVNE : BOOL;
	VonkajsieValcovanie_AKTIVNE : BOOL;
	CasVypnutiaHydrauliky : TON;
	Stav_ServaREADY : BOOL;
	SC_Oddelovac : SequenceControlTyp;
	Oddelovac_Automat : BOOL;
	Oddelovac_Manual : BOOL;
	Oddelovac_Reset : BOOL;
	Oddelovac_PoINIT : BOOL;
	Oddelovac_KoniecVyroby : BOOL;
	Oddelovac_KoniecCyklu : BOOL;
	SC_ZdvihRotora : SequenceControlTyp;
	ZdvihRotora_Automat : BOOL;
	ZdvihRotora_Manual : BOOL;
	ZdvihRotora_Reset : BOOL;
	ZdvihRotora_PoINIT : BOOL;
	ZdvihRotora_KoniecVyroby : BOOL;
	ZdvihRotora_KoniecCyklu : BOOL;
	SC_VstupnyManipulator : SequenceControlTyp;
	VstupManipulator_Automat : BOOL;
	VstupManipulator_Manual : BOOL;
	VstupManipulator_Reset : BOOL;
	VstupManipulator_PoINIT : BOOL;
	VstupManipulator_KoniecVyroby : BOOL;
	VstupManipulator_KoniecCyklu : BOOL;
	VstupManipulator_RychlJoggingu : REAL;
	VstupManipulator_RychlostPolohov : REAL;
	VstupManipul_Rychlost_MM_s : REAL;
END_VAR
VAR RETAIN
	VstupManipul_RychlostJog_MM_s : REAL;
END_VAR
VAR
	VstupManipulator_HomingOK : BOOL;
	VstupManipulator_AktualPozMM : REAL;
	VstupManipulator_ZadanaPozMM : REAL;
	VstupManipulator_PojazdVPOZICI : BOOL;
	VstupManipulator_PrebiehaHoming : BOOL;
	VstupManipulator_PojazdHOME : BOOL;
	VstupManipulator_UkoncilCyklus : BOOL;
END_VAR
VAR RETAIN
	VstupManipulator_Drzi_NG_Kus : BOOL;
END_VAR
VAR
	VstupManipulator_OdobralRotor : BOOL;
	SC_Stol : SequenceControlTyp;
	Stol_Automat : BOOL;
	Stol_Manual : BOOL;
	Stol_Reset : BOOL;
	Stol_PoINIT : BOOL;
	Stol_KoniecVyroby : BOOL;
	Stol_KoniecCyklu : BOOL;
	Stol_PrebehloOtocenie : BOOL;
	Stol_BlokovanieOtacania : BOOL;
	Stol_CakaNaVstupnyManipulator : BOOL;
	Stol_CakaNaStrihanie : BOOL;
	Stol_CakaNaRazenie : BOOL;
	Stol_CakaNaValcovanie : BOOL;
	Stol_CakaNaMeranie : BOOL;
	Stol_CakaNaVystupnyManipulator : BOOL;
	Stol_NG_KusNaStole : BOOL;
	Stol_OdoberNG_Kus : BOOL;
	Stol_StavPrazdnyStol : BOOL;
	Stol_RR_OtacajVPRED : BOOL;
	Stol_RR_OtacajVZAD : BOOL;
END_VAR
VAR RETAIN
	Stol_Pozicia_1 : USINT; (*Pozicia stola pod meranim  0 - neznamy kus, 1 - kus OK, 2 - kus NG *)
	Stol_Pozicia_2 : USINT; (*Pozícia medzi meranim a výstupným manipulátorom    0 - neznamy kus, 1 - kus OK, 2 - kus NG *)
	Stol_Pozicia_3 : USINT; (*Pozícia pod výstupným manipulátorom     0 - neznamy kus, 1 - kus OK, 2 - kus NG *)
END_VAR
VAR
	SC_Strihanie : SequenceControlTyp;
	Strihanie_Automat : BOOL;
	Strihanie_Manual : BOOL;
	Strihanie_Reset : BOOL;
	Strihanie_PoINIT : BOOL;
	Strihanie_KoniecVyroby : BOOL;
	Strihanie_KoniecCyklu : BOOL;
	Strihanie_UkoncilCyklus : BOOL;
	Strihanie_SpustiRazenie : BOOL;
	Strihanie_RR_Centrovanie_OTVOR : BOOL;
	Strihanie_RR_Centrovanie_ZATVOR : BOOL;
	SC_Razenie : SequenceControlTyp;
	Razenie_Automat : BOOL;
	Razenie_Manual : BOOL;
	Razenie_Reset : BOOL;
	Razenie_PoINIT : BOOL;
	Razenie_KoniecVyroby : BOOL;
	Razenie_KoniecCyklu : BOOL;
	Razenie_UkoncilCyklus : BOOL;
	SC_Valcovanie : SequenceControlTyp;
	Valcovanie_Automat : BOOL;
	Valcovanie_Manual : BOOL;
	Valcovanie_Reset : BOOL;
	Valcovanie_PoINIT : BOOL;
	Valcovanie_KoniecVyroby : BOOL;
	Valcovanie_KoniecCyklu : BOOL;
	Valcovanie_ServoRychlJoggingu : REAL;
	Valcovanie_ServoRychlostPolohov : REAL;
	Valcovanie_Rychlost_MM_s : REAL;
END_VAR
VAR RETAIN
	Valcovanie_RychlostJog_MM_s : REAL;
END_VAR
VAR
	Valcovanie_HomingOK : BOOL;
	Valcovanie_AktualPozMM : REAL;
	Valcovanie_ZadanaPozMM : REAL;
	Valcovanie_ZdvihVPOZICI : BOOL;
	Valcovanie_PrebiehaHoming : BOOL;
	Valcovanie_ZdvihHOME : BOOL;
	Valcovanie_FM_RozbehRampa : UINT; (*0.1*)
	Valcovanie_FM_DobehRampa : UINT; (*0.1*)
	Valcovanie_FM_RychlostOtac_Hz : INT;
	Valcovanie_UkoncilCyklus : BOOL;
	CasValcovania_ms : TIME;
	SC_Valcovanie2 : SequenceControlTyp;
	Valcovanie2_Automat : BOOL;
	Valcovanie2_Manual : BOOL;
	Valcovanie2_Reset : BOOL;
	Valcovanie2_PoINIT : BOOL;
	Valcovanie2_KoniecVyroby : BOOL;
	Valcovanie2_KoniecCyklu : BOOL;
END_VAR
VAR RETAIN
	Valcovanie2_ServoJoggRychl_MM_s : REAL;
	Valcovanie2_ServoPracRychl1_MM_s : REAL; (*Rýchlosť priblíženia*)
	Valcovanie2_ServoPracRychl2_MM_s : REAL; (*Rýchlosť valcovania*)
	Valcovanie2_MomentPritlaku_Nm : REAL;
END_VAR
VAR
	Valcovanie2_HomingOK : BOOL;
	Valcovanie2_AktualPozMM : REAL;
END_VAR
VAR RETAIN
	Valcovanie2_ZadanaPozMM : REAL;
	Valcovanie2_ZadanaPozSTART_MM : REAL; (*Čakacia pozícia pod stolom*)
END_VAR
VAR
	Valcovanie2_ZdvihVPOZICI : BOOL;
	Valcovanie2_PrebiehaHoming : BOOL;
	Valcovanie2_ZdvihHOME : BOOL;
END_VAR
VAR RETAIN
	Valcovanie2_FM_RozbehRampa_s : REAL;
	Valcovanie2_FM_DobehRampa_s : REAL;
	Valcovanie2_FM_RychlostOtac_Hz : REAL;
END_VAR
VAR
	Valcovanie2_UkoncilCyklus : BOOL;
END_VAR
VAR RETAIN
	Valcovanie2_CasValcovania_s : REAL;
	Valcovanie2_CasStrekuOleja_s : REAL;
	Valcovanie2_PocetCyklStrekuOleja : USINT;
END_VAR
VAR
	Valcovanie2_DavkaOleja : BOOL;
	SC_Meranie : SequenceControlTyp;
	Meranie_Automat : BOOL;
	Meranie_Manual : BOOL;
	Meranie_Reset : BOOL;
	Meranie_PoINIT : BOOL;
	Meranie_KoniecVyroby : BOOL;
	Meranie_KoniecCyklu : BOOL;
	Meranie_FM_RozbehRampa : UINT;
	Meranie_FM_DobehRampa : UINT; (*0.1*)
	Meranie_FM_RychlostOtac_Hz : INT; (*0.1*)
	Meranie_UkoncilCyklus : BOOL;
	Meranie_ObsluhaRozhodla : BOOL;
	SC_VystupnyManipulator : SequenceControlTyp;
	VystupManipulator_Automat : BOOL;
	VystupManipulator_Manual : BOOL;
	VystupManipulator_Reset : BOOL;
	VystupManipulator_PoINIT : BOOL;
	VystupManipulator_KoniecVyroby : BOOL;
	VystupManipulator_KoniecCyklu : BOOL;
	VystupManipulator_RychlJoggingu : REAL;
	VystupManipulator_RychlostPoloho : REAL;
	VystupManipul_Rychlost_MM_s : REAL;
END_VAR
VAR RETAIN
	VystupManipul_RychlostJog_MM_s : REAL;
END_VAR
VAR
	VystupManipulator_HomingOK : BOOL;
	VystupManipulator_AktualPozMM : REAL;
	VystupManipulator_ZadanaPozMM : REAL;
	VystupManipulator_PojazdVPOZICI : BOOL;
	VystupManipulator_PrebiehaHoming : BOOL;
	VystupManipulator_PojazdHOME : BOOL;
	VystupManipulator_UkoncilCyklus : BOOL;
	VystupManipulator_OdoberNGKus : BOOL;
	VystupManipulator_Drzi_OK_Kus : BOOL;
	VystupManipulator_Drzi_NG_Kus : BOOL;
	SC_VystupnyOdsuvac : SequenceControlTyp;
	VystupOdsuvac_Automat : BOOL;
	VystupOdsuvac_Manual : BOOL;
	VystupOdsuvac_Reset : BOOL;
	VystupOdsuvac_PoINIT : BOOL;
	VystupOdsuvac_KoniecVyroby : BOOL;
	VystupOdsuvac_KoniecCyklu : BOOL;
	VystupOdsuvac_CakaNaKusy : BOOL;
	VystupOdsuvac_KusyVlozene : BOOL;
END_VAR
(*************Vizualizacia***********************)
VAR
	CisloAktualnejObrazovky : USINT;
	CisloZadanejObrazovky : USINT;
	BlikanieTlacitkaStartZariadenia : BOOL;
	TP_ModraLEDResetCS : USINT;
	TP_ModraLEDResetOplotenia : USINT;
	TP_ZamkniTlacStartAutomat : USINT;
	TP_ZamkniTlacUkoncenieVyroby : USINT;
	TP_ZamkniTlacKoniecCyklu : USINT;
	TP_ZobrazHlasenieResetZariadenia : USINT;
	TP_ZobrazTlacitkoSetup : USINT;
	TP_ZobrazTlacitkoAlarmy : USINT;
	TP_ZobrazTlacitkoHome : USINT;
	TP_ZobrazTlacitkoSpat : USINT;
	TP_ZobrazHlasenieDoprNG_Plny : USINT;
	TP_ZobrazHlasenieDoprOK_Plny : USINT;
	TP_ZobrazHlasenieNizkaHladOleja : USINT;
	TP_ZobrazHlasenieZamkyVyblokov : USINT;
	TP_ZamkniTlacitkoOtacanieStola : USINT;
	TP_ZamkniTlacitkoHomingServ : USINT;
	TP_ZamkniTlacitkoOvladanieZamkov : USINT;
	TP_ZamkniTlacitkoOvladanieBZ1 : USINT;
	TP_ZamkniTlacitkoOvladanieBZ2 : USINT;
	TP_ZamkniTlacitkoOvladanieBZ3 : USINT;
	TP_ZamkniTlacitkoOvladanieBZ4 : USINT;
	TP_ZamkniTlacitkoOvladanieBZ5 : USINT;
	TP_ZamkniTlacitkoOvladanieBZ6 : USINT;
	TP_ZamkniTlacitkoRezimAutomat : USINT;
	TP_ZamkniTlacitkoRezimRevork : USINT;
	TP_ZamkniTlacitkaAktivValcovania : USINT;
	TP_ZamkniTlacitkoRezimManual : USINT;
	TP_ZamkniTlacitkaZamkovOplotenia : USINT;
	TP_ZamkniTlacitkoServis : USINT;
	TP_VstupManip_ZamkniTlacPojazdu : USINT;
	TP_Strihanie_ZamkniZdvihRotora : USINT;
	TP_Valcovanie_ZamkniZdvihRotora : USINT;
	TP_Valcovanie_ZamkniZdvihServa : USINT;
	TP_Valcovanie2_ZamkniZdvihServa : USINT;
	TP_Valcovanie2_ZamkniZostupServa : USINT;
	TP_Valcovanie2_ZamkniHomeServa : USINT;
	TP_Valcovanie2_ZamkniOtacVPRED : USINT;
	TP_Valcovanie2_ZamkniOtacVZAD : USINT;
	TP_Razenie_ZamkniZdvihRotora : USINT;
	TP_Stol_ZamkniOtacanie : USINT;
	TP_Stol_Centrovanie_VYSUN : BOOL;
	TP_Stol_Centrovanie_ZASUN : BOOL;
	TP_Meranie_ZamkniZdvihRotora : USINT;
	TP_VystupManip_ZamkniTlacPojazdu : USINT;
	TP_VystOdsuvac_ZamkniTlacVysunut : USINT;
END_VAR
VAR RETAIN
	TP_VstupManip_PoziciaOdoberania : REAL; (*v mm*)
	TP_VstupManip_PoziciaUkladania : REAL; (*v mm*)
	TP_VstupManip_RychlostPojazdu : REAL; (*v mm/s*)
	TP_Razenie_CasRazenia : REAL; (*v s*)
	TP_Valcovanie_PoziciaVnorenia : REAL; (*v mm*)
	TP_Valcovanie_RychlostZdvihu : REAL; (*v mm/s*)
	TP_Valcovanie_RychlostOtacania : INT; (*v Hz*)
	TP_Valcovanie_CasStrekuOleja : REAL; (*v s*)
	TP_Valcovanie_PocetCyklPredStrek : UINT;
	TP_Meranie_RychlostOtacania : INT; (*v Hz*)
	TP_Meranie_CasMerania : REAL; (*v s*)
	TP_VystupManip_PoziciaOdoberania : REAL; (*v mm*)
	TP_VystupManip_PoziciaUklad_OK : REAL; (*v mm*)
	TP_VystupManip_PoziciaUklad_NG : REAL; (*v mm*)
	TP_VystupManip_RychlostPojazdu : REAL; (*v mm/s*)
END_VAR
VAR
	TP_Zariadenie_TaktTime : REAL;
	TP_ZamkniParametreUrovenOperator : USINT;
	TP_ZamkniParametreUrovenServisak : USINT;
END_VAR
VAR RETAIN
	TP_CasValcovania_s : REAL; (*v sek*)
END_VAR
VAR
	Slider : UINT;
	StavOddelovaca : USINT;
	StavZdvihuRotora : USINT;
	StavVstupnehoManipulatora : USINT;
	StavStola : USINT;
	StavStrihania : USINT;
	StavRazenia : USINT;
	StavValcovania : USINT;
	StavValcovania2 : USINT;
	StavMerania : USINT;
	StavVystupnehoManipulatora : USINT;
	StavVystupnehoOdsuvaca : USINT;
	StavOperatora : USINT;
	TEST : BOOL;
END_VAR
(****Komunikácie medzi PLC*********)
VAR
	ModBus_Input1 : UINT;
	ModBus_Input2 : UINT;
	ModBus_Input3 : UINT;
	ModBus_Input4 : UINT;
	ModBus_Input5 : UINT;
	ModBus_Output1 : UINT;
	ModBus_Output2 : UINT;
	ModBus_Output3 : UINT;
	ModBus_Output4 : UINT;
	ModBus_Output5 : UINT;
END_VAR
(****Komunikácie medzi PLC*********)
VAR
	Stol : StolStruc;
	Vyrazanie : VyrazanieStruc;
END_VAR
```

### Package Logical/Libraries - Global libraries

### Library Logical/Libraries/IecCheck (IEC)
Depends on: sys_lib, AsBrStr

#### IecCheck.fun - Exported functions and function blocks
```iecst
FUNCTION CheckDivSint : SINT (* Check divisor for SINT division *)
	VAR_INPUT
		divisor : SINT;
	END_VAR
END_FUNCTION

FUNCTION CheckDivUsint : USINT (* Check divisor for USINT division *)
	VAR_INPUT
		divisor : USINT;
	END_VAR
END_FUNCTION

FUNCTION CheckDivInt : INT (* Check divisor for INT division *)
	VAR_INPUT
		divisor : INT;
	END_VAR
END_FUNCTION

FUNCTION CheckDivUint : UINT (* Check divisor for UINT division *)
	VAR_INPUT
		divisor : UINT;
	END_VAR
END_FUNCTION

FUNCTION CheckDivDint : DINT (* Check divisor for DINT division *)
	VAR_INPUT
		divisor : DINT;
	END_VAR
END_FUNCTION

FUNCTION CheckDivUdint : UDINT (* Check divisor for UDINT division *)
	VAR_INPUT
		divisor : UDINT;
	END_VAR
END_FUNCTION

FUNCTION CheckDivReal : REAL (* Check divisor for REAL division *)
	VAR_INPUT
		divisor : REAL;
	END_VAR
END_FUNCTION

FUNCTION CheckDivLReal : LREAL (* Check divisor for LREAL division, not available for SG3 and SGC *)
	VAR_INPUT
		divisor : LREAL;
	END_VAR
END_FUNCTION

FUNCTION CheckBounds : DINT (* Check range for array access *)
	VAR_INPUT
		index : DINT;
		lower : DINT;
		upper : DINT;
	END_VAR
END_FUNCTION

FUNCTION CheckRange : DINT (* Check range for enumeration *)
	VAR_INPUT
		value : DINT;
		lower : DINT;
		upper : DINT;
	END_VAR
END_FUNCTION

FUNCTION CheckSignedSubrange : DINT (* Check range for subrange of signed data types *)
	VAR_INPUT
		value : DINT;
		lower : DINT;
		upper : DINT;
	END_VAR
END_FUNCTION

FUNCTION CheckUnsignedSubrange : UDINT (* Check range for subrange of unsigned data types *)
	VAR_INPUT
		value : UDINT;
		lower : UDINT;
		upper : UDINT;
	END_VAR
END_FUNCTION

FUNCTION CheckReadAccess : UDINT (* Check address when reading dynamic variables *)
	VAR_INPUT
		address : UDINT;
	END_VAR
END_FUNCTION

FUNCTION CheckWriteAccess : UDINT (* Check address when writing dynamic variables *)
	VAR_INPUT
		address : UDINT;
	END_VAR
END_FUNCTION

FUNCTION MakeEntry : UDINT (* Makes an entry (log book entry) in the error log book *)
	VAR
		taskname : STRING[30];
		group : USINT;
		status_name : UINT;
		out_text : STRING[80];
	END_VAR
	VAR_INPUT
		number : UINT;
		index : DINT;
		text : STRING[50];
	END_VAR
END_FUNCTION
```

#### IecCheck.st - Implementation file
```iecst
(* Check divisor for SINT division *)
FUNCTION CheckDivSint
	IF divisor=0 THEN
		CheckDivSint:=1;
		MakeEntry(55555,divisor,'CheckDivSint');
	ELSE
		CheckDivSint:=divisor;
	END_IF
END_FUNCTION

(* Check divisor for USINT division *)
FUNCTION CheckDivUsint
	IF divisor=0 THEN
		CheckDivUsint:=1;
		MakeEntry(55555,divisor,'CheckDivUsint');
	ELSE
		CheckDivUsint:=divisor;
	END_IF
END_FUNCTION

(* Check divisor for INT division *)
FUNCTION CheckDivInt
	IF divisor=0 THEN
		CheckDivInt:=1;
		MakeEntry(55555,divisor,'CheckDivInt');
	ELSE
		CheckDivInt:=divisor;
	END_IF
END_FUNCTION

(* Check divisor for UINT division *)
FUNCTION CheckDivUint
	IF divisor=0 THEN
		CheckDivUint:=1;
		MakeEntry(55555,divisor,'CheckDivUint');
	ELSE
		CheckDivUint:=divisor;
	END_IF
END_FUNCTION

(* Check divisor for DINT division *)
FUNCTION CheckDivDint
	IF divisor=0 THEN
		CheckDivDint:=1;
		MakeEntry(55555,divisor,'CheckDivDint');
	ELSE
		CheckDivDint:=divisor;
	END_IF
END_FUNCTION

(* Check divisor for UDINT division *)
FUNCTION CheckDivUdint
	IF divisor=0 THEN
		CheckDivUdint:=1;
		MakeEntry(55555,divisor,'CheckDivUdint');
	ELSE
		CheckDivUdint:=divisor;
	END_IF
END_FUNCTION

(* Check divisor for REAL division *)
FUNCTION CheckDivReal
	IF divisor=0 THEN
		CheckDivReal:=1;
		MakeEntry(55555,0,'CheckDivReal');
	ELSE
		CheckDivReal:=divisor;
	END_IF
END_FUNCTION

(* Check divisor for LREAL division *)
FUNCTION CheckDivLReal
	IF divisor=0 THEN
		CheckDivLReal:=1;
		MakeEntry(55555,0,'CheckDivLReal');
	ELSE
		CheckDivLReal:=divisor;
	END_IF
END_FUNCTION

(* Check range for array access *)
FUNCTION CheckBounds
	IF index < lower THEN
		CheckBounds := lower;
		MakeEntry(55555,index,'CheckBounds');
	ELSIF index > upper THEN
		CheckBounds := upper;
		MakeEntry(55555,index,'CheckBounds');
	ELSE
		CheckBounds := index;
	END_IF
END_FUNCTION

(* Check range for enumeration *)
FUNCTION CheckRange
	IF value < lower THEN
		CheckRange := lower;
		MakeEntry(55555,value,'CheckRange');
	ELSIF value > upper THEN
		CheckRange := upper;
		MakeEntry(55555,value,'CheckRange');
	ELSE
		CheckRange := value;
	END_IF
END_FUNCTION

(* Check range for subrange of signed data types *)
FUNCTION CheckSignedSubrange
	IF value < lower THEN
		CheckSignedSubrange := lower;
		MakeEntry(55555,value,'CheckSignedSubrange');
	ELSIF value > upper THEN
		CheckSignedSubrange := upper;
		MakeEntry(55555,value,'CheckSignedSubrange');
	ELSE
		CheckSignedSubrange := value;
	END_IF
END_FUNCTION

(* Check range for subrange of unsigned data types *)
FUNCTION CheckUnsignedSubrange
	IF value < lower THEN
		CheckUnsignedSubrange := lower;
		MakeEntry(55555,value,'CheckUnsignedSubrange');
	ELSIF value > upper THEN
		CheckUnsignedSubrange := upper;
		MakeEntry(55555,value,'CheckUnsignedSubrange');
	ELSE
		CheckUnsignedSubrange := value;
	END_IF
END_FUNCTION

(* Check address when reading dynamic variables *)
FUNCTION CheckReadAccess
	IF address=0 THEN
		(* TODO: Insert an appropriate code, see AutomationStudio help for further information *)
		MakeEntry(55555,address,'Read from NULL');
	END_IF

	CheckReadAccess:=0;
END_FUNCTION

(* Check address when writing dynamic variables *)
FUNCTION CheckWriteAccess
	IF address=0 THEN
		(* TODO: Insert an appropriate code, see AutomationStudio help for further information *)
		MakeEntry(55555,address,'Write to NULL');
	END_IF

	CheckWriteAccess:=0;
END_FUNCTION

(* Makes an entry (log book entry) in the error log book *)
FUNCTION MakeEntry
		status_name := ST_name(0,ADR(taskname),ADR(group));

		brsstrcpy(ADR(out_text),ADR(text));
		brsstrcat(ADR(out_text),ADR(' > in task > '));
  		brsstrcat(ADR(out_text),ADR(taskname));
		MakeEntry := ADR(out_text);
		ERRxfatal(number,index,ADR(out_text));
END_FUNCTION
```

### Library Logical/Libraries/SC (IEC)

#### Types.typ - Exported data types
```iecst
TYPE
	SequenceControlTyp : 	STRUCT
		StepName : STRING[80];
		Step : UINT;
		Switch1 : BOOL;
		Switch2 : BOOL;
		Switch3 : BOOL;
		ResetStep : BOOL;
		LastStep : BOOL;
		IdleTime : TON;
		AlarmTime : TON;
	END_STRUCT;
END_TYPE
```

#### SC.fun - Exported functions and function blocks
```iecst
FUNCTION SequenceControl : BOOL
	VAR_IN_OUT
		SC : SequenceControlTyp;
	END_VAR
END_FUNCTION
```

#### SequenceControl.st
```iecst
(* TODO: Add your comment here *)
FUNCTION SequenceControl

	IF SC.ResetStep THEN
		brsmemset(ADR(SC.StepName),0,SIZEOF(SC.StepName));
		SC.Switch1:= FALSE;
		SC.Switch2:= FALSE;
		SC.Switch3:= FALSE;
		SC.IdleTime.IN:= FALSE;
		SC.AlarmTime.IN:= FALSE;
		SC.ResetStep:= FALSE;
	END_IF

	IF SC.LastStep THEN
		brsmemset(ADR(SC.StepName),0,SIZEOF(SC.StepName));
		SC.Switch1:= FALSE;
		SC.Switch2:= FALSE;
		SC.Switch3:= FALSE;
		SC.IdleTime.IN:= FALSE;
		SC.AlarmTime.IN:= FALSE;
		SC.Step:= 0;
		SC.LastStep:= FALSE;
	END_IF

	//Volanie časovačov//
	SC.AlarmTime();
	SC.IdleTime();

END_FUNCTION
```

### Library Logical/Libraries/AxisLib (ANSIC, version 1.10.6) - Motion Library
Depends on: AsBrStr, Acp10_MC, NcGlobal

#### AxisLib.typ - Exported data types
```iecst
(* ********************************************************************
  * COPYRIGHT -- Bernecker + Rainer
  ********************************************************************
  * Author: Milan Jun
  * Created: May 28, 2014
  *********************************************************************)
(**)
(*Axes structures*)

TYPE
	AxisCommand_type : 	STRUCT  (*Command structure for single axis.*)
		power : BOOL; (*Switch on the controller.*)
		home : BOOL; (*Reference axis.*)
		moveAbsolute : BOOL; (*Move to a defined position.*)
		moveVelocity : BOOL; (*Move with a defined speed.*)
		moveAdditive : BOOL; (*Move a defined distance.*)
		moveTorqueControl : BOOL; (*Move torque control.*)
		moveVelocityControl : BOOL; (*Move cyclic velocity*)
		moveJogPos : BOOL; (*Move jog positive.*)
		moveJogNeg : BOOL; (*Move jog negative.*)
		halt : BOOL; (*Stop every active movement on the axis.*)
		stop : BOOL; (*Stop every active movement on the axis as long as is set.*)
		errorAck : BOOL; (*Error acknowledge.*)
		autoInicialization : BOOL; (*Automatic inicialization ( power-home-ack error ).*)
	END_STRUCT;
	AxisParameterVelocityCtrl_type : 	STRUCT  (*Specific structure for velocity control fb*)
		cyclicVelocity : REAL; (*Velocity for MoveVelocity-Command.*)
		cyclicVelocityCorrection : REAL;
		cyclicTorque : REAL; (*Velocity for MoveVelocity-Command.*)
		TorqueMode : USINT; (*VelocityControl torque mode*)
		sCtrlKv : REAL; (*VelocityControl proporcional part*)
		sCtrlTn : REAL; (*VelocityControl integration part*)
		initSctrl : BOOL;
	END_STRUCT;
	AxisParameter_type : 	STRUCT  (*Parameter structure.*)
		acc : REAL; (*Acceleration for commanded movements.*)
		dec : REAL; (*Deceleration for commanded movements.*)
		axis : UDINT; (*Axis reference.*)
		position : REAL; (*Target position for MoveAbsolute-Command.*)
		distance : REAL; (*Distance for MoveAdditive-Command.*)
		velocity : REAL; (*Velocity for MoveVelocity-Command.*)
		direction : USINT; (*Direction for commanded movements.*)
		torque : REAL;
		torqueRamp : REAL;
		homePos : REAL; (*Target position for referencing the axis.*)
		homeMode : USINT; (*Homing mode.*)
		blockMoveVelocity : BOOL; (*Block in move velocity step*)
		velocityControl : AxisParameterVelocityCtrl_type;
		velocityJog : REAL; (*Velocity joggingu*)
	END_STRUCT;
	AxisStatus_type : 	STRUCT  (*Status structure.*)
		ActTorque : REAL; (*Actual position of the axis.*)
		ActPosition : REAL; (*Actual position of the axis.*)
		ActVelocity : REAL; (*Actual velocity of the axis.*)
		DriveStatus : MC_DRIVESTATUS_TYP; (*Actual status of the axis.*)
	END_STRUCT;
	AxisState_type : 	STRUCT  (*Axis state structure.*)
		Disabled : BOOL; (*If set, axis is in state Disabled.*)
		StandStill : BOOL; (*If set, axis is in state StandsStill.*)
		Homing : BOOL; (*if set, axis is in state Homing.*)
		Stopping : BOOL; (*If set, axis is in state Stopping.*)
		DiscreteMotion : BOOL; (*If set, axis is in state DiscreteMotion.*)
		ContinuousMotion : BOOL; (*If set, axis is in state ContinuousMotion.*)
		SynchronizedMotion : BOOL; (*If set, axis is in state SynchronizedMotion.*)
		ErrorStop : BOOL; (*If set, axis is in state ErrorStop.*)
	END_STRUCT;
	AxisError_type : 	STRUCT  (*Error structure.*)
		AxisErrorCount : UINT; (*Number of active axis errors.*)
		AxisWarningCount : UINT; (*Number of active axis warinings.*)
		FunctionBlockErrorCount : UINT; (*Number of active function block errors.*)
		ErrorRecord : MC_ERRORRECORD_REF; (*Error record information.*)
		ErrorText : ARRAY[0..3]OF STRING[79]; (*Description of first active error or warning.*)
		ErrorID : UDINT;
		ErrorStatus : USINT;
	END_STRUCT;
	AxisInternal_type : 	STRUCT  (*Axis internal type, all used function blocks and internal variables*)
		MC_BR_ReadDriveStatus_0 : MC_BR_ReadDriveStatus;
		MC_ReadStatus_0 : MC_ReadStatus;
		MC_ReadActualPosition_0 : MC_ReadActualPosition;
		MC_ReadActualTorque_0 : MC_ReadActualTorque;
		MC_ReadActualVelocity_0 : MC_ReadActualVelocity;
		MC_ReadAxisError_0 : MC_ReadAxisError;
		MC_Reset_0 : MC_Reset;
		MC_Power_0 : MC_Power;
		MC_Home_0 : MC_Home;
		MC_Halt_0 : MC_Halt;
		MC_Stop_0 : MC_Stop;
		MC_MoveAdditive_0 : MC_MoveAdditive;
		MC_MoveAbsolute_0 : MC_MoveAbsolute;
		MC_MoveVelocity_0 : MC_MoveVelocity;
		MC_BR_VelocityControl_0 : MC_BR_VelocityControl;
		MC_TorqueControl_0 : MC_TorqueControl;
		MC_BR_BrakeOperation_0 : MC_BR_BrakeOperation;
		MC_BR_ReadParID_0 : MC_BR_ReadParID;
		MC_BR_WriteParID_0 : MC_BR_WriteParID;
		AxisReadStep : USINT;
		AxisStep : AxisStateStep_Enum;
		InitStep : AxisStateInitStep_Enum;
		errorOld : UDINT;
		TimeCheck : UINT;
		switch2 : BOOL;
		switch1 : BOOL;
		brakeMode : BOOL;
	END_STRUCT;
END_TYPE

(**)
(*Axes enumeration*)

TYPE
	AxisStateStep_Enum :
		(
		AXISSTATE_WAIT := 0,
		AXISSTATE_POWER_ON := 1,
		AXISSTATE_READY := 2,
		AXISSTATE_HOME := 3,
		AXISSTATE_HALT := 4,
		AXISSTATE_STOP := 5,
		AXISSTATE_MOVE_ABSOLUTE := 6,
		AXISSTATE_MOVE_ADDITIVE := 7,
		AXISSTATE_MOVE_VELOCITY := 8,
		AXISSTATE_MOVE_JOGPOS := 9,
		AXISSTATE_MOVE_TORQUE_CONTROL := 10,
		AXISSTATE_MOVE_JOGNEG := 11,
		AXISSTATE_ERROR_AXIS := 14,
		AXISSTATE_ERROR := 15,
		AXISSTATE_ERROR_RESET := 16,
		AXISSTATE_MOVE_VELOCITY_CONTROL := 20
		);
	AxisStateInitStep_Enum :
		(
		STATE_INIT := 0,
		STATE_WATCH := 1,
		STATE_SWITCHON := 2,
		STATE_HOME := 3,
		STATE_ERROR_HANDLE := 4
		);
END_TYPE

(**)
(*Axis extension*)

TYPE
	AxisExtensionCommand_type : 	STRUCT
		cmdRstEncoder : BOOL;
		cmdReadTemp : BOOL;
		cmdReadCurrent : BOOL;
		cmdReadLagError : BOOL;
		cmdBrakeToggle : BOOL;
		cmdBrake : BOOL;
		cmdUnbrake : BOOL;
		cmdGetHwInfo : BOOL;
	END_STRUCT;
	AxisExtensionParameter_type : 	STRUCT
		axis : UDINT; (*Axis reference.*)
	END_STRUCT;
	AxisExtensionStatus_type : 	STRUCT
		ActMotorTemp : REAL; (*Actual motor temperature*)
		ActMotorCurrent : REAL; (*Actual motor current*)
		ActLagError : REAL;
		HardwareInfo : MC_HARDWARE_INFO_REF;
	END_STRUCT;
	AxisExtensionInternal_type : 	STRUCT
		MC_BR_ReadParID_0 : MC_BR_ReadParID;
		MC_BR_WriteParID_0 : MC_BR_WriteParID;
		MC_BR_BrakeOperation_0 : MC_BR_BrakeOperation;
		MC_BR_GetHardwareInfo_0 : MC_BR_GetHardwareInfo;
		brakeMode : BOOL;
		AxisReadStep : USINT;
	END_STRUCT;
END_TYPE
```

#### AxisLib.var - Exported constants
```iecst
(* ********************************************************************
  * COPYRIGHT -- Bernecker + Rainer
  ********************************************************************
  * Author: Milan Jun
  * Created: May 28, 2014
  *********************************************************************)
VAR CONSTANT
	ret : UDINT := 0;
END_VAR
```

#### AxisLib.fun - Axis functions/function blocks
```iecst
(* ********************************************************************
  * COPYRIGHT -- Bernecker + Rainer
  ********************************************************************
  * Author: Milan Jun
  * Created: May 28, 2014
  *********************************************************************)

FUNCTION_BLOCK Axis (*Axis motion*) (*$GROUP=User*)
	VAR_INPUT
		enable : BOOL; (*Enables/Disables the function block.*)
		cmd : AxisCommand_type; (*Axis commands.*)
		par : AxisParameter_type; (*Axis parameters.*)
	END_VAR
	VAR_OUTPUT
		active : BOOL; (*Function block is active.*)
		busy : BOOL; (*Function block is busy.*)
		error : BOOL; (*Function block is an error.*)
		errorCount : UDINT; (*Error counter.*)
		errorID : UDINT; (*Error id.*)
		errorText : ARRAY[0..3] OF STRING[79]; (*Error text.*)
		status : AxisStatus_type;
		state : AxisState_type;
	END_VAR
	VAR
		internal : AxisInternal_type;
	END_VAR
END_FUNCTION_BLOCK

FUNCTION_BLOCK AxisExtension (* *) (*$GROUP=User,$CAT=User,$GROUPICON=User.png,$CATICON=User.png*)
	VAR_INPUT
		enable : BOOL;
		cmd : AxisExtensionCommand_type;
		par : AxisExtensionParameter_type;
	END_VAR
	VAR_OUTPUT
		active : BOOL;
		status : AxisExtensionStatus_type;
		errorID : UDINT; (*Error id.*)
	END_VAR
	VAR
		internal : AxisExtensionInternal_type;
	END_VAR
END_FUNCTION_BLOCK
```
